Fanuc TP program (LS listing): 190220_hosenrohr_oV5.ls

/PROG  190220_hosenrohr_oV5
/ATTR
COMMENT	= "19-02-22 10:03:29";
PROG_SIZE	= 0;
DEFAULT_GROUP	= 1, 1, *, *, *;
/APPL
    ARC Welding Equipment: 1, *, *, *, *;
/MN
   1:  CALL HOME_ALL;
   1:  UFRAME_NUM = 1;
   1:  UTOOL_NUM = 3;
   1:  COL GUARD ADJUST 150;
   1:  ! -- Layer/Ebene 207 -- !;
   1:  PR[91] = PR[90];
   1:  PR[GP1:91,1] = PR[GP1:90,1] + -0.916;
   1:  PR[GP1:91,2] = PR[GP1:90,2] + 48.907;
   1:  PR[GP1:91,3] = PR[GP1:90,3] + 126.575;
   1:  !Sicherheitspunkt!;
   1:  PR[92] = PR[91];
   1:  PR[92] = PR[GP1:92,3] + 50;
   1:J PR[92];
   1:  !Schweissanfang anfahren!;
   1:L PR[91] R[100]mm/sec CNT100;
   1:  CALL LASER_DRAHT_START;
   1:  PR[GP1:91,1] = PR[GP1:90,1] + -12.234;
   1:  PR[GP1:91,2] = PR[GP1:90,2] + 47.505;
   1:L PR[91] R[100]mm/sec CNT100;
   1:  PR[GP1:91,1] = PR[GP1:90,1] + -13.167;
   1:  PR[GP1:91,2] = PR[GP1:90,2] + 47.191;
   1:L PR[91] R[100]mm/sec CNT100;
   1:  PR[GP1:91,1] = PR[GP1:90,1] + -23.762;
   1:  PR[GP1:91,2] = PR[GP1:90,2] + 43.085;
   1:L PR[91] R[100]mm/sec CNT100;
   1:  PR[GP1:91,1] = PR[GP1:90,1] + -24.573;
   1:  PR[GP1:91,2] = PR[GP1:90,2] + 42.437;
   1:L PR[91] R[100]mm/sec CNT100;
   1:  PR[GP1:91,1] = PR[GP1:90,1] + -33.854;
   1:  PR[GP1:91,2] = PR[GP1:90,2] + 35.865;
   1:L PR[91] R[100]mm/sec CNT100;
   1:  PR[GP1:91,1] = PR[GP1:90,1] + -41.983;
   1:  PR[GP1:91,2] = PR[GP1:90,2] + 26.074;
   1:L PR[91] R[100]mm/sec CNT100;
   1:  PR[GP1:91,1] = PR[GP1:90,1] + -42.514;
   1:  PR[GP1:91,2] = PR[GP1:90,2] + 25.188;
   1:L PR[91] R[100]mm/sec CNT100;
   1:  PR[GP1:91,1] = PR[GP1:90,1] + -47.649;
   1:  PR[GP1:91,2] = PR[GP1:90,2] + 13.555;
   1:L PR[91] R[100]mm/sec CNT100;
   1:  PR[GP1:91,1] = PR[GP1:90,1] + -47.838;
   1:  PR[GP1:91,2] = PR[GP1:90,2] + 12.520;
   1:L PR[91] R[100]mm/sec CNT100;
   1:  PR[GP1:91,1] = PR[GP1:90,1] + -49.592;
   1:  PR[GP1:91,2] = PR[GP1:90,2] + -0.059;
   1:L PR[91] R[100]mm/sec CNT100;
   1:  PR[GP1:91,1] = PR[GP1:90,1] + -49.406;
   1:  PR[GP1:91,2] = PR[GP1:90,2] + -1.079;
   1:L PR[91] R[100]mm/sec CNT100;
   1:  PR[GP1:91,1] = PR[GP1:90,1] + -47.644;
   1:  PR[GP1:91,2] = PR[GP1:90,2] + -13.710;
   1:L PR[91] R[100]mm/sec CNT100;
   1:  PR[GP1:91,1] = PR[GP1:90,1] + -42.514;
   1:  PR[GP1:91,2] = PR[GP1:90,2] + -25.332;
   1:L PR[91] R[100]mm/sec CNT100;
   1:  PR[GP1:91,1] = PR[GP1:90,1] + -41.983;
   1:  PR[GP1:91,2] = PR[GP1:90,2] + -26.218;
   1:L PR[91] R[100]mm/sec CNT100;
   1:  PR[GP1:91,1] = PR[GP1:90,1] + -33.843;
   1:  PR[GP1:91,2] = PR[GP1:90,2] + -36.023;
   1:L PR[91] R[100]mm/sec CNT100;
   1:  PR[GP1:91,1] = PR[GP1:90,1] + -33.064;
   1:  PR[GP1:91,2] = PR[GP1:90,2] + -36.648;
   1:L PR[91] R[100]mm/sec CNT100;
   1:  PR[GP1:91,1] = PR[GP1:90,1] + -23.779;
   1:  PR[GP1:91,2] = PR[GP1:90,2] + -43.223;
   1:L PR[91] R[100]mm/sec CNT100;
   1:  PR[GP1:91,1] = PR[GP1:90,1] + -13.167;
   1:  PR[GP1:91,2] = PR[GP1:90,2] + -47.335;
   1:L PR[91] R[100]mm/sec CNT100;
   1:  PR[GP1:91,1] = PR[GP1:90,1] + -12.234;
   1:  PR[GP1:91,2] = PR[GP1:90,2] + -47.649;
   1:L PR[91] R[100]mm/sec CNT100;
   1:  PR[GP1:91,1] = PR[GP1:90,1] + -0.916;
   1:  PR[GP1:91,2] = PR[GP1:90,2] + -49.051;
   1:L PR[91] R[100]mm/sec CNT100;
   1:  PR[GP1:91,1] = PR[GP1:90,1] + 0.047;
   1:  PR[GP1:91,2] = PR[GP1:90,2] + -49.031;
   1:L PR[91] R[100]mm/sec CNT100;
   1:  PR[GP1:91,1] = PR[GP1:90,1] + 1.125;
   1:  PR[GP1:91,2] = PR[GP1:90,2] + -49.051;
   1:L PR[91] R[100]mm/sec CNT100;
   1:  PR[GP1:91,1] = PR[GP1:90,1] + 12.446;
   1:  PR[GP1:91,2] = PR[GP1:90,2] + -47.650;
   1:L PR[91] R[100]mm/sec CNT100;
   1:  PR[GP1:91,1] = PR[GP1:90,1] + 13.378;
   1:  PR[GP1:91,2] = PR[GP1:90,2] + -47.335;
   1:L PR[91] R[100]mm/sec CNT100;
   1:  PR[GP1:91,1] = PR[GP1:90,1] + 23.975;
   1:  PR[GP1:91,2] = PR[GP1:90,2] + -43.229;
   1:L PR[91] R[100]mm/sec CNT100;
   1:  PR[GP1:91,1] = PR[GP1:90,1] + 24.786;
   1:  PR[GP1:91,2] = PR[GP1:90,2] + -42.581;
   1:L PR[91] R[100]mm/sec CNT100;
   1:  PR[GP1:91,1] = PR[GP1:90,1] + 34.069;
   1:  PR[GP1:91,2] = PR[GP1:90,2] + -36.008;
   1:L PR[91] R[100]mm/sec CNT100;
   1:  PR[GP1:91,1] = PR[GP1:90,1] + 42.197;
   1:  PR[GP1:91,2] = PR[GP1:90,2] + -26.217;
   1:L PR[91] R[100]mm/sec CNT100;
   1:  PR[GP1:91,1] = PR[GP1:90,1] + 42.727;
   1:  PR[GP1:91,2] = PR[GP1:90,2] + -25.331;
   1:L PR[91] R[100]mm/sec CNT100;
   1:  PR[GP1:91,1] = PR[GP1:90,1] + 47.863;
   1:  PR[GP1:91,2] = PR[GP1:90,2] + -13.699;
   1:L PR[91] R[100]mm/sec CNT100;
   1:  PR[GP1:91,1] = PR[GP1:90,1] + 48.051;
   1:  PR[GP1:91,2] = PR[GP1:90,2] + -12.663;
   1:L PR[91] R[100]mm/sec CNT100;
   1:  PR[GP1:91,1] = PR[GP1:90,1] + 49.806;
   1:  PR[GP1:91,2] = PR[GP1:90,2] + -0.085;
   1:L PR[91] R[100]mm/sec CNT100;
   1:  PR[GP1:91,1] = PR[GP1:90,1] + 49.619;
   1:  PR[GP1:91,2] = PR[GP1:90,2] + 0.935;
   1:L PR[91] R[100]mm/sec CNT100;
   1:  PR[GP1:91,1] = PR[GP1:90,1] + 47.857;
   1:  PR[GP1:91,2] = PR[GP1:90,2] + 13.566;
   1:L PR[91] R[100]mm/sec CNT100;
   1:  PR[GP1:91,1] = PR[GP1:90,1] + 42.727;
   1:  PR[GP1:91,2] = PR[GP1:90,2] + 25.187;
   1:L PR[91] R[100]mm/sec CNT100;
   1:  PR[GP1:91,1] = PR[GP1:90,1] + 42.197;
   1:  PR[GP1:91,2] = PR[GP1:90,2] + 26.073;
   1:L PR[91] R[100]mm/sec CNT100;
   1:  PR[GP1:91,1] = PR[GP1:90,1] + 34.058;
   1:  PR[GP1:91,2] = PR[GP1:90,2] + 35.878;
   1:L PR[91] R[100]mm/sec CNT100;
   1:  PR[GP1:91,1] = PR[GP1:90,1] + 33.278;
   1:  PR[GP1:91,2] = PR[GP1:90,2] + 36.503;
   1:L PR[91] R[100]mm/sec CNT100;
   1:  PR[GP1:91,1] = PR[GP1:90,1] + 23.992;
   1:  PR[GP1:91,2] = PR[GP1:90,2] + 43.079;
   1:L PR[91] R[100]mm/sec CNT100;
   1:  PR[GP1:91,1] = PR[GP1:90,1] + 13.378;
   1:  PR[GP1:91,2] = PR[GP1:90,2] + 47.192;
   1:L PR[91] R[100]mm/sec CNT100;
   1:  PR[GP1:91,1] = PR[GP1:90,1] + 12.445;
   1:  PR[GP1:91,2] = PR[GP1:90,2] + 47.506;
   1:L PR[91] R[100]mm/sec CNT100;
   1:  PR[GP1:91,1] = PR[GP1:90,1] + 1.125;
   1:  PR[GP1:91,2] = PR[GP1:90,2] + 48.907;
   1:L PR[91] R[100]mm/sec CNT100;
   1:  PR[GP1:91,1] = PR[GP1:90,1] + 0.047;
   1:  PR[GP1:91,2] = PR[GP1:90,2] + 48.887;
   1:L PR[91] R[100]mm/sec CNT100;
   1:  ! -- Layer/Ebene 208 -- !;
   1:  PR[91] = PR[90];
   1:  PR[GP1:91,1] = PR[GP1:90,1] + -0.545;
   1:  PR[GP1:91,2] = PR[GP1:90,2] + 49.055;
   1:  PR[GP1:91,3] = PR[GP1:90,3] + 127.185;
   1:L PR[91] R[100]mm/sec CNT100;
   1:  PR[GP1:91,1] = PR[GP1:90,1] + -12.137;
   1:  PR[GP1:91,2] = PR[GP1:90,2] + 47.619;
   1:L PR[91] R[100]mm/sec CNT100;
   1:  PR[GP1:91,1] = PR[GP1:90,1] + -12.717;
   1:  PR[GP1:91,2] = PR[GP1:90,2] + 47.424;
   1:L PR[91] R[100]mm/sec CNT100;
   1:  PR[GP1:91,1] = PR[GP1:90,1] + -23.582;
   1:  PR[GP1:91,2] = PR[GP1:90,2] + 43.214;
   1:L PR[91] R[100]mm/sec CNT100;
   1:  PR[GP1:91,1] = PR[GP1:90,1] + -24.086;
   1:  PR[GP1:91,2] = PR[GP1:90,2] + 42.811;
   1:L PR[91] R[100]mm/sec CNT100;
   1:  PR[GP1:91,1] = PR[GP1:90,1] + -33.614;
   1:  PR[GP1:91,2] = PR[GP1:90,2] + 36.064;
   1:L PR[91] R[100]mm/sec CNT100;
   1:  PR[GP1:91,1] = PR[GP1:90,1] + -41.959;
   1:  PR[GP1:91,2] = PR[GP1:90,2] + 26.012;
   1:L PR[91] R[100]mm/sec CNT100;
   1:  PR[GP1:91,1] = PR[GP1:90,1] + -42.288;
   1:  PR[GP1:91,2] = PR[GP1:90,2] + 25.463;
   1:L PR[91] R[100]mm/sec CNT100;
   1:  PR[GP1:91,1] = PR[GP1:90,1] + -47.564;
   1:  PR[GP1:91,2] = PR[GP1:90,2] + 13.512;
   1:L PR[91] R[100]mm/sec CNT100;
   1:  PR[GP1:91,1] = PR[GP1:90,1] + -47.681;
   1:  PR[GP1:91,2] = PR[GP1:90,2] + 12.871;
   1:L PR[91] R[100]mm/sec CNT100;
   1:  PR[GP1:91,1] = PR[GP1:90,1] + -49.484;
   1:  PR[GP1:91,2] = PR[GP1:90,2] + -0.059;
   1:L PR[91] R[100]mm/sec CNT100;
   1:  PR[GP1:91,1] = PR[GP1:90,1] + -49.369;
   1:  PR[GP1:91,2] = PR[GP1:90,2] + -0.690;
   1:L PR[91] R[100]mm/sec CNT100;
   1:  PR[GP1:91,1] = PR[GP1:90,1] + -47.559;
   1:  PR[GP1:91,2] = PR[GP1:90,2] + -13.667;
   1:L PR[91] R[100]mm/sec CNT100;
   1:  PR[GP1:91,1] = PR[GP1:90,1] + -42.288;
   1:  PR[GP1:91,2] = PR[GP1:90,2] + -25.607;
   1:L PR[91] R[100]mm/sec CNT100;
   1:  PR[GP1:91,1] = PR[GP1:90,1] + -41.959;
   1:  PR[GP1:91,2] = PR[GP1:90,2] + -26.156;
   1:L PR[91] R[100]mm/sec CNT100;
   1:  PR[GP1:91,1] = PR[GP1:90,1] + -33.602;
   1:  PR[GP1:91,2] = PR[GP1:90,2] + -36.222;
   1:L PR[91] R[100]mm/sec CNT100;
   1:  PR[GP1:91,1] = PR[GP1:90,1] + -33.120;
   1:  PR[GP1:91,2] = PR[GP1:90,2] + -36.609;
   1:L PR[91] R[100]mm/sec CNT100;
   1:  PR[GP1:91,1] = PR[GP1:90,1] + -23.599;
   1:  PR[GP1:91,2] = PR[GP1:90,2] + -43.351;
   1:L PR[91] R[100]mm/sec CNT100;
   1:  PR[GP1:91,1] = PR[GP1:90,1] + -12.717;
   1:  PR[GP1:91,2] = PR[GP1:90,2] + -47.568;
   1:L PR[91] R[100]mm/sec CNT100;
   1:  PR[GP1:91,1] = PR[GP1:90,1] + -12.138;
   1:  PR[GP1:91,2] = PR[GP1:90,2] + -47.763;
   1:L PR[91] R[100]mm/sec CNT100;
   1:  PR[GP1:91,1] = PR[GP1:90,1] + -0.545;
   1:  PR[GP1:91,2] = PR[GP1:90,2] + -49.199;
   1:L PR[91] R[100]mm/sec CNT100;
   1:  PR[GP1:91,1] = PR[GP1:90,1] + 0.067;
   1:  PR[GP1:91,2] = PR[GP1:90,2] + -49.186;
   1:L PR[91] R[100]mm/sec CNT100;
   1:  PR[GP1:91,1] = PR[GP1:90,1] + 0.754;
   1:  PR[GP1:91,2] = PR[GP1:90,2] + -49.199;
   1:L PR[91] R[100]mm/sec CNT100;
   1:  PR[GP1:91,1] = PR[GP1:90,1] + 12.349;
   1:  PR[GP1:91,2] = PR[GP1:90,2] + -47.764;
   1:L PR[91] R[100]mm/sec CNT100;
   1:  PR[GP1:91,1] = PR[GP1:90,1] + 12.928;
   1:  PR[GP1:91,2] = PR[GP1:90,2] + -47.569;
   1:L PR[91] R[100]mm/sec CNT100;
   1:  PR[GP1:91,1] = PR[GP1:90,1] + 23.795;
   1:  PR[GP1:91,2] = PR[GP1:90,2] + -43.358;
   1:L PR[91] R[100]mm/sec CNT100;
   1:  PR[GP1:91,1] = PR[GP1:90,1] + 24.299;
   1:  PR[GP1:91,2] = PR[GP1:90,2] + -42.955;
   1:L PR[91] R[100]mm/sec CNT100;
   1:  PR[GP1:91,1] = PR[GP1:90,1] + 33.829;
   1:  PR[GP1:91,2] = PR[GP1:90,2] + -36.207;
   1:L PR[91] R[100]mm/sec CNT100;
   1:  PR[GP1:91,1] = PR[GP1:90,1] + 42.173;
   1:  PR[GP1:91,2] = PR[GP1:90,2] + -26.155;
   1:L PR[91] R[100]mm/sec CNT100;
   1:  PR[GP1:91,1] = PR[GP1:90,1] + 42.501;
   1:  PR[GP1:91,2] = PR[GP1:90,2] + -25.607;
   1:L PR[91] R[100]mm/sec CNT100;
   1:  PR[GP1:91,1] = PR[GP1:90,1] + 47.777;
   1:  PR[GP1:91,2] = PR[GP1:90,2] + -13.655;
   1:L PR[91] R[100]mm/sec CNT100;
   1:  PR[GP1:91,1] = PR[GP1:90,1] + 47.894;
   1:  PR[GP1:91,2] = PR[GP1:90,2] + -13.014;
   1:L PR[91] R[100]mm/sec CNT100;
   1:  PR[GP1:91,1] = PR[GP1:90,1] + 49.698;
   1:  PR[GP1:91,2] = PR[GP1:90,2] + -0.085;
   1:L PR[91] R[100]mm/sec CNT100;
   1:  PR[GP1:91,1] = PR[GP1:90,1] + 49.582;
   1:  PR[GP1:91,2] = PR[GP1:90,2] + 0.546;
   1:L PR[91] R[100]mm/sec CNT100;
   1:  PR[GP1:91,1] = PR[GP1:90,1] + 47.772;
   1:  PR[GP1:91,2] = PR[GP1:90,2] + 13.523;
   1:L PR[91] R[100]mm/sec CNT100;
   1:  PR[GP1:91,1] = PR[GP1:90,1] + 42.501;
   1:  PR[GP1:91,2] = PR[GP1:90,2] + 25.463;
   1:L PR[91] R[100]mm/sec CNT100;
   1:  PR[GP1:91,1] = PR[GP1:90,1] + 42.173;
   1:  PR[GP1:91,2] = PR[GP1:90,2] + 26.011;
   1:L PR[91] R[100]mm/sec CNT100;
   1:  PR[GP1:91,1] = PR[GP1:90,1] + 33.817;
   1:  PR[GP1:91,2] = PR[GP1:90,2] + 36.077;
   1:L PR[91] R[100]mm/sec CNT100;
   1:  PR[GP1:91,1] = PR[GP1:90,1] + 33.334;
   1:  PR[GP1:91,2] = PR[GP1:90,2] + 36.464;
   1:L PR[91] R[100]mm/sec CNT100;
   1:  PR[GP1:91,1] = PR[GP1:90,1] + 23.812;
   1:  PR[GP1:91,2] = PR[GP1:90,2] + 43.207;
   1:L PR[91] R[100]mm/sec CNT100;
   1:  PR[GP1:91,1] = PR[GP1:90,1] + 12.928;
   1:  PR[GP1:91,2] = PR[GP1:90,2] + 47.425;
   1:L PR[91] R[100]mm/sec CNT100;
   1:  PR[GP1:91,1] = PR[GP1:90,1] + 12.349;
   1:  PR[GP1:91,2] = PR[GP1:90,2] + 47.620;
   1:L PR[91] R[100]mm/sec CNT100;
   1:  PR[GP1:91,1] = PR[GP1:90,1] + 0.754;
   1:  PR[GP1:91,2] = PR[GP1:90,2] + 49.056;
   1:L PR[91] R[100]mm/sec CNT100;
   1:  PR[GP1:91,1] = PR[GP1:90,1] + 0.067;
   1:  PR[GP1:91,2] = PR[GP1:90,2] + 49.042;
   1:L PR[91] R[100]mm/sec CNT100;
   1:  ! -- Layer/Ebene 209 -- !;
   1:  PR[91] = PR[90];
   1:  PR[GP1:91,1] = PR[GP1:90,1] + -12.041;
   1:  PR[GP1:91,2] = PR[GP1:90,2] + 47.733;
   1:  PR[GP1:91,3] = PR[GP1:90,3] + 127.795;
   1:L PR[91] R[100]mm/sec CNT100;
   1:  PR[GP1:91,1] = PR[GP1:90,1] + -12.266;
   1:  PR[GP1:91,2] = PR[GP1:90,2] + 47.657;
   1:L PR[91] R[100]mm/sec CNT100;
   1:  PR[GP1:91,1] = PR[GP1:90,1] + -23.402;
   1:  PR[GP1:91,2] = PR[GP1:90,2] + 43.342;
   1:L PR[91] R[100]mm/sec CNT100;
   1:  PR[GP1:91,1] = PR[GP1:90,1] + -23.600;
   1:  PR[GP1:91,2] = PR[GP1:90,2] + 43.184;
   1:L PR[91] R[100]mm/sec CNT100;
   1:  PR[GP1:91,1] = PR[GP1:90,1] + -33.373;
   1:  PR[GP1:91,2] = PR[GP1:90,2] + 36.263;
   1:L PR[91] R[100]mm/sec CNT100;
   1:  PR[GP1:91,1] = PR[GP1:90,1] + -41.935;
   1:  PR[GP1:91,2] = PR[GP1:90,2] + 25.950;
   1:L PR[91] R[100]mm/sec CNT100;
   1:  PR[GP1:91,1] = PR[GP1:90,1] + -42.062;
   1:  PR[GP1:91,2] = PR[GP1:90,2] + 25.739;
   1:L PR[91] R[100]mm/sec CNT100;
   1:  PR[GP1:91,1] = PR[GP1:90,1] + -47.479;
   1:  PR[GP1:91,2] = PR[GP1:90,2] + 13.468;
   1:L PR[91] R[100]mm/sec CNT100;
   1:  PR[GP1:91,1] = PR[GP1:90,1] + -47.524;
   1:  PR[GP1:91,2] = PR[GP1:90,2] + 13.221;
   1:L PR[91] R[100]mm/sec CNT100;
   1:  PR[GP1:91,1] = PR[GP1:90,1] + -49.376;
   1:  PR[GP1:91,2] = PR[GP1:90,2] + -0.059;
   1:L PR[91] R[100]mm/sec CNT100;
   1:  PR[GP1:91,1] = PR[GP1:90,1] + -49.332;
   1:  PR[GP1:91,2] = PR[GP1:90,2] + -0.302;
   1:L PR[91] R[100]mm/sec CNT100;
   1:  PR[GP1:91,1] = PR[GP1:90,1] + -47.474;
   1:  PR[GP1:91,2] = PR[GP1:90,2] + -13.624;
   1:L PR[91] R[100]mm/sec CNT100;
   1:  PR[GP1:91,1] = PR[GP1:90,1] + -42.062;
   1:  PR[GP1:91,2] = PR[GP1:90,2] + -25.883;
   1:L PR[91] R[100]mm/sec CNT100;
   1:  PR[GP1:91,1] = PR[GP1:90,1] + -41.935;
   1:  PR[GP1:91,2] = PR[GP1:90,2] + -26.094;
   1:L PR[91] R[100]mm/sec CNT100;
   1:  PR[GP1:91,1] = PR[GP1:90,1] + -33.362;
   1:  PR[GP1:91,2] = PR[GP1:90,2] + -36.421;
   1:L PR[91] R[100]mm/sec CNT100;
   1:  PR[GP1:91,1] = PR[GP1:90,1] + -33.176;
   1:  PR[GP1:91,2] = PR[GP1:90,2] + -36.570;
   1:L PR[91] R[100]mm/sec CNT100;
   1:  PR[GP1:91,1] = PR[GP1:90,1] + -23.418;
   1:  PR[GP1:91,2] = PR[GP1:90,2] + -43.480;
   1:L PR[91] R[100]mm/sec CNT100;
   1:  PR[GP1:91,1] = PR[GP1:90,1] + -12.266;
   1:  PR[GP1:91,2] = PR[GP1:90,2] + -47.801;
   1:L PR[91] R[100]mm/sec CNT100;
   1:  PR[GP1:91,1] = PR[GP1:90,1] + -12.041;
   1:  PR[GP1:91,2] = PR[GP1:90,2] + -47.877;
   1:L PR[91] R[100]mm/sec CNT100;
   1:  PR[GP1:91,1] = PR[GP1:90,1] + -0.168;
   1:  PR[GP1:91,2] = PR[GP1:90,2] + -49.348;
   1:L PR[91] R[100]mm/sec CNT100;
   1:  PR[GP1:91,1] = PR[GP1:90,1] + 0.377;
   1:L PR[91] R[100]mm/sec CNT100;
   1:  PR[GP1:91,1] = PR[GP1:90,1] + 12.252;
   1:  PR[GP1:91,2] = PR[GP1:90,2] + -47.878;
   1:L PR[91] R[100]mm/sec CNT100;
   1:  PR[GP1:91,1] = PR[GP1:90,1] + 12.478;
   1:  PR[GP1:91,2] = PR[GP1:90,2] + -47.802;
   1:L PR[91] R[100]mm/sec CNT100;
   1:  PR[GP1:91,1] = PR[GP1:90,1] + 23.615;
   1:  PR[GP1:91,2] = PR[GP1:90,2] + -43.486;
   1:L PR[91] R[100]mm/sec CNT100;
   1:  PR[GP1:91,1] = PR[GP1:90,1] + 23.812;
   1:  PR[GP1:91,2] = PR[GP1:90,2] + -43.328;
   1:L PR[91] R[100]mm/sec CNT100;
   1:  PR[GP1:91,1] = PR[GP1:90,1] + 33.588;
   1:  PR[GP1:91,2] = PR[GP1:90,2] + -36.406;
   1:L PR[91] R[100]mm/sec CNT100;
   1:  PR[GP1:91,1] = PR[GP1:90,1] + 42.149;
   1:  PR[GP1:91,2] = PR[GP1:90,2] + -26.093;
   1:L PR[91] R[100]mm/sec CNT100;
   1:  PR[GP1:91,1] = PR[GP1:90,1] + 42.275;
   1:  PR[GP1:91,2] = PR[GP1:90,2] + -25.882;
   1:L PR[91] R[100]mm/sec CNT100;
   1:  PR[GP1:91,1] = PR[GP1:90,1] + 47.692;
   1:  PR[GP1:91,2] = PR[GP1:90,2] + -13.612;
   1:L PR[91] R[100]mm/sec CNT100;
   1:  PR[GP1:91,1] = PR[GP1:90,1] + 47.737;
   1:  PR[GP1:91,2] = PR[GP1:90,2] + -13.365;
   1:L PR[91] R[100]mm/sec CNT100;
   1:  PR[GP1:91,1] = PR[GP1:90,1] + 49.589;
   1:  PR[GP1:91,2] = PR[GP1:90,2] + -0.085;
   1:L PR[91] R[100]mm/sec CNT100;
   1:  PR[GP1:91,1] = PR[GP1:90,1] + 49.545;
   1:  PR[GP1:91,2] = PR[GP1:90,2] + 0.158;
   1:L PR[91] R[100]mm/sec CNT100;
   1:  PR[GP1:91,1] = PR[GP1:90,1] + 47.687;
   1:  PR[GP1:91,2] = PR[GP1:90,2] + 13.480;
   1:L PR[91] R[100]mm/sec CNT100;
   1:  PR[GP1:91,1] = PR[GP1:90,1] + 42.275;
   1:  PR[GP1:91,2] = PR[GP1:90,2] + 25.738;
   1:L PR[91] R[100]mm/sec CNT100;
   1:  PR[GP1:91,1] = PR[GP1:90,1] + 42.149;
   1:  PR[GP1:91,2] = PR[GP1:90,2] + 25.949;
   1:L PR[91] R[100]mm/sec CNT100;
   1:  PR[GP1:91,1] = PR[GP1:90,1] + 33.577;
   1:  PR[GP1:91,2] = PR[GP1:90,2] + 36.276;
   1:L PR[91] R[100]mm/sec CNT100;
   1:  PR[GP1:91,1] = PR[GP1:90,1] + 33.390;
   1:  PR[GP1:91,2] = PR[GP1:90,2] + 36.425;
   1:L PR[91] R[100]mm/sec CNT100;
   1:  PR[GP1:91,1] = PR[GP1:90,1] + 23.631;
   1:  PR[GP1:91,2] = PR[GP1:90,2] + 43.336;
   1:L PR[91] R[100]mm/sec CNT100;
   1:  PR[GP1:91,1] = PR[GP1:90,1] + 12.477;
   1:  PR[GP1:91,2] = PR[GP1:90,2] + 47.658;
   1:L PR[91] R[100]mm/sec CNT100;
   1:  PR[GP1:91,1] = PR[GP1:90,1] + 12.252;
   1:  PR[GP1:91,2] = PR[GP1:90,2] + 47.734;
   1:L PR[91] R[100]mm/sec CNT100;
   1:  PR[GP1:91,1] = PR[GP1:90,1] + 0.377;
   1:  PR[GP1:91,2] = PR[GP1:90,2] + 49.204;
   1:L PR[91] R[100]mm/sec CNT100;
   1:  PR[GP1:91,1] = PR[GP1:90,1] + -0.168;
   1:L PR[91] R[100]mm/sec CNT100;
   1:  ! -- Layer/Ebene 210 -- !;
   1:  PR[91] = PR[90];
   1:  PR[GP1:91,1] = PR[GP1:90,1] + -11.979;
   1:  PR[GP1:91,2] = PR[GP1:90,2] + 47.821;
   1:  PR[GP1:91,3] = PR[GP1:90,3] + 128.405;
   1:L PR[91] R[100]mm/sec CNT100;
   1:  PR[GP1:91,1] = PR[GP1:90,1] + -23.226;
   1:  PR[GP1:91,2] = PR[GP1:90,2] + 43.462;
   1:L PR[91] R[100]mm/sec CNT100;
   1:  PR[GP1:91,1] = PR[GP1:90,1] + -23.300;
   1:  PR[GP1:91,2] = PR[GP1:90,2] + 43.425;
   1:L PR[91] R[100]mm/sec CNT100;
   1:  PR[GP1:91,1] = PR[GP1:90,1] + -33.152;
   1:  PR[GP1:91,2] = PR[GP1:90,2] + 36.449;
   1:L PR[91] R[100]mm/sec CNT100;
   1:  PR[GP1:91,1] = PR[GP1:90,1] + -33.209;
   1:  PR[GP1:91,2] = PR[GP1:90,2] + 36.392;
   1:L PR[91] R[100]mm/sec CNT100;
   1:  PR[GP1:91,1] = PR[GP1:90,1] + -41.871;
   1:  PR[GP1:91,2] = PR[GP1:90,2] + 25.958;
   1:L PR[91] R[100]mm/sec CNT100;
   1:  PR[GP1:91,1] = PR[GP1:90,1] + -47.397;
   1:  PR[GP1:91,2] = PR[GP1:90,2] + 13.461;
   1:L PR[91] R[100]mm/sec CNT100;
   1:  PR[GP1:91,1] = PR[GP1:90,1] + -49.288;
   1:  PR[GP1:91,2] = PR[GP1:90,2] + -0.072;
   1:L PR[91] R[100]mm/sec CNT100;
   1:  PR[GP1:91,1] = PR[GP1:90,1] + -47.411;
   1:  PR[GP1:91,2] = PR[GP1:90,2] + -13.529;
   1:L PR[91] R[100]mm/sec CNT100;
   1:  PR[GP1:91,1] = PR[GP1:90,1] + -47.399;
   1:  PR[GP1:91,2] = PR[GP1:90,2] + -13.600;
   1:L PR[91] R[100]mm/sec CNT100;
   1:  PR[GP1:91,1] = PR[GP1:90,1] + -41.871;
   1:  PR[GP1:91,2] = PR[GP1:90,2] + -26.102;
   1:L PR[91] R[100]mm/sec CNT100;
   1:  PR[GP1:91,1] = PR[GP1:90,1] + -33.209;
   1:  PR[GP1:91,2] = PR[GP1:90,2] + -36.536;
   1:L PR[91] R[100]mm/sec CNT100;
   1:  PR[GP1:91,1] = PR[GP1:90,1] + -33.152;
   1:  PR[GP1:91,2] = PR[GP1:90,2] + -36.592;
   1:L PR[91] R[100]mm/sec CNT100;
   1:  PR[GP1:91,1] = PR[GP1:90,1] + -23.300;
   1:  PR[GP1:91,2] = PR[GP1:90,2] + -43.569;
   1:L PR[91] R[100]mm/sec CNT100;
   1:  PR[GP1:91,1] = PR[GP1:90,1] + -23.226;
   1:  PR[GP1:91,2] = PR[GP1:90,2] + -43.606;
   1:L PR[91] R[100]mm/sec CNT100;
   1:  PR[GP1:91,1] = PR[GP1:90,1] + -11.979;
   1:  PR[GP1:91,2] = PR[GP1:90,2] + -47.965;
   1:L PR[91] R[100]mm/sec CNT100;
   1:  PR[GP1:91,1] = PR[GP1:90,1] + 0.105;
   1:  PR[GP1:91,2] = PR[GP1:90,2] + -49.467;
   1:L PR[91] R[100]mm/sec CNT100;
   1:  PR[GP1:91,1] = PR[GP1:90,1] + 12.190;
   1:  PR[GP1:91,2] = PR[GP1:90,2] + -47.965;
   1:L PR[91] R[100]mm/sec CNT100;
   1:  PR[GP1:91,1] = PR[GP1:90,1] + 23.439;
   1:  PR[GP1:91,2] = PR[GP1:90,2] + -43.606;
   1:L PR[91] R[100]mm/sec CNT100;
   1:  PR[GP1:91,1] = PR[GP1:90,1] + 23.513;
   1:  PR[GP1:91,2] = PR[GP1:90,2] + -43.569;
   1:L PR[91] R[100]mm/sec CNT100;
   1:  PR[GP1:91,1] = PR[GP1:90,1] + 33.367;
   1:  PR[GP1:91,2] = PR[GP1:90,2] + -36.591;
   1:L PR[91] R[100]mm/sec CNT100;
   1:  PR[GP1:91,1] = PR[GP1:90,1] + 33.421;
   1:  PR[GP1:91,2] = PR[GP1:90,2] + -36.536;
   1:L PR[91] R[100]mm/sec CNT100;
   1:  PR[GP1:91,1] = PR[GP1:90,1] + 42.085;
   1:  PR[GP1:91,2] = PR[GP1:90,2] + -26.101;
   1:L PR[91] R[100]mm/sec CNT100;
   1:  PR[GP1:91,1] = PR[GP1:90,1] + 47.610;
   1:  PR[GP1:91,2] = PR[GP1:90,2] + -13.605;
   1:L PR[91] R[100]mm/sec CNT100;
   1:  PR[GP1:91,1] = PR[GP1:90,1] + 49.501;
   1:  PR[GP1:91,2] = PR[GP1:90,2] + -0.072;
   1:L PR[91] R[100]mm/sec CNT100;
   1:  PR[GP1:91,1] = PR[GP1:90,1] + 47.610;
   1:  PR[GP1:91,2] = PR[GP1:90,2] + 13.461;
   1:L PR[91] R[100]mm/sec CNT100;
   1:  PR[GP1:91,1] = PR[GP1:90,1] + 42.085;
   1:  PR[GP1:91,2] = PR[GP1:90,2] + 25.957;
   1:L PR[91] R[100]mm/sec CNT100;
   1:  PR[GP1:91,1] = PR[GP1:90,1] + 33.421;
   1:  PR[GP1:91,2] = PR[GP1:90,2] + 36.393;
   1:L PR[91] R[100]mm/sec CNT100;
   1:  PR[GP1:91,1] = PR[GP1:90,1] + 33.367;
   1:  PR[GP1:91,2] = PR[GP1:90,2] + 36.447;
   1:L PR[91] R[100]mm/sec CNT100;
   1:  PR[GP1:91,1] = PR[GP1:90,1] + 23.513;
   1:  PR[GP1:91,2] = PR[GP1:90,2] + 43.425;
   1:L PR[91] R[100]mm/sec CNT100;
   1:  PR[GP1:91,1] = PR[GP1:90,1] + 23.439;
   1:  PR[GP1:91,2] = PR[GP1:90,2] + 43.462;
   1:L PR[91] R[100]mm/sec CNT100;
   1:  PR[GP1:91,1] = PR[GP1:90,1] + 12.181;
   1:  PR[GP1:91,2] = PR[GP1:90,2] + 47.825;
   1:L PR[91] R[100]mm/sec CNT100;
   1:  PR[GP1:91,1] = PR[GP1:90,1] + 12.099;
   1:  PR[GP1:91,2] = PR[GP1:90,2] + 47.838;
   1:L PR[91] R[100]mm/sec CNT100;
   1:  PR[GP1:91,1] = PR[GP1:90,1] + 0.105;
   1:  PR[GP1:91,2] = PR[GP1:90,2] + 49.323;
   1:L PR[91] R[100]mm/sec CNT100;
   1:  ! -- Layer/Ebene 211 -- !;
   1:  PR[91] = PR[90];
   1:  PR[GP1:91,1] = PR[GP1:90,1] + -11.144;
   1:  PR[GP1:91,2] = PR[GP1:90,2] + 47.930;
   1:  PR[GP1:91,3] = PR[GP1:90,3] + 129.015;
   1:L PR[91] R[100]mm/sec CNT100;
   1:  PR[GP1:91,1] = PR[GP1:90,1] + -12.168;
   1:  PR[GP1:91,2] = PR[GP1:90,2] + 47.768;
   1:L PR[91] R[100]mm/sec CNT100;
   1:  PR[GP1:91,1] = PR[GP1:90,1] + -22.726;
   1:  PR[GP1:91,2] = PR[GP1:90,2] + 43.676;
   1:L PR[91] R[100]mm/sec CNT100;
   1:  PR[GP1:91,1] = PR[GP1:90,1] + -23.649;
   1:  PR[GP1:91,2] = PR[GP1:90,2] + 43.205;
   1:L PR[91] R[100]mm/sec CNT100;
   1:  PR[GP1:91,1] = PR[GP1:90,1] + -32.890;
   1:  PR[GP1:91,2] = PR[GP1:90,2] + 36.662;
   1:L PR[91] R[100]mm/sec CNT100;
   1:  PR[GP1:91,1] = PR[GP1:90,1] + -33.621;
   1:  PR[GP1:91,2] = PR[GP1:90,2] + 35.931;
   1:L PR[91] R[100]mm/sec CNT100;
   1:  PR[GP1:91,1] = PR[GP1:90,1] + -41.756;
   1:  PR[GP1:91,2] = PR[GP1:90,2] + 26.132;
   1:L PR[91] R[100]mm/sec CNT100;
   1:  PR[GP1:91,1] = PR[GP1:90,1] + -42.222;
   1:  PR[GP1:91,2] = PR[GP1:90,2] + 25.217;
   1:L PR[91] R[100]mm/sec CNT100;
   1:  PR[GP1:91,1] = PR[GP1:90,1] + -47.364;
   1:  PR[GP1:91,2] = PR[GP1:90,2] + 13.569;
   1:L PR[91] R[100]mm/sec CNT100;
   1:  PR[GP1:91,1] = PR[GP1:90,1] + -49.126;
   1:  PR[GP1:91,2] = PR[GP1:90,2] + 0.936;
   1:L PR[91] R[100]mm/sec CNT100;
   1:  PR[GP1:91,1] = PR[GP1:90,1] + -49.287;
   1:  PR[GP1:91,2] = PR[GP1:90,2] + -0.078;
   1:L PR[91] R[100]mm/sec CNT100;
   1:  PR[GP1:91,1] = PR[GP1:90,1] + -47.527;
   1:  PR[GP1:91,2] = PR[GP1:90,2] + -12.694;
   1:L PR[91] R[100]mm/sec CNT100;
   1:  PR[GP1:91,1] = PR[GP1:90,1] + -47.366;
   1:  PR[GP1:91,2] = PR[GP1:90,2] + -13.708;
   1:L PR[91] R[100]mm/sec CNT100;
   1:  PR[GP1:91,1] = PR[GP1:90,1] + -42.222;
   1:  PR[GP1:91,2] = PR[GP1:90,2] + -25.361;
   1:L PR[91] R[100]mm/sec CNT100;
   1:  PR[GP1:91,1] = PR[GP1:90,1] + -41.756;
   1:  PR[GP1:91,2] = PR[GP1:90,2] + -26.276;
   1:L PR[91] R[100]mm/sec CNT100;
   1:  PR[GP1:91,1] = PR[GP1:90,1] + -33.621;
   1:  PR[GP1:91,2] = PR[GP1:90,2] + -36.075;
   1:L PR[91] R[100]mm/sec CNT100;
   1:  PR[GP1:91,1] = PR[GP1:90,1] + -32.890;
   1:  PR[GP1:91,2] = PR[GP1:90,2] + -36.806;
   1:L PR[91] R[100]mm/sec CNT100;
   1:  PR[GP1:91,1] = PR[GP1:90,1] + -23.649;
   1:  PR[GP1:91,2] = PR[GP1:90,2] + -43.349;
   1:L PR[91] R[100]mm/sec CNT100;
   1:  PR[GP1:91,1] = PR[GP1:90,1] + -22.726;
   1:  PR[GP1:91,2] = PR[GP1:90,2] + -43.820;
   1:L PR[91] R[100]mm/sec CNT100;
   1:  PR[GP1:91,1] = PR[GP1:90,1] + -12.177;
   1:  PR[GP1:91,2] = PR[GP1:90,2] + -47.908;
   1:L PR[91] R[100]mm/sec CNT100;
   1:  PR[GP1:91,1] = PR[GP1:90,1] + -0.909;
   1:  PR[GP1:91,2] = PR[GP1:90,2] + -49.304;
   1:L PR[91] R[100]mm/sec CNT100;
   1:  PR[GP1:91,1] = PR[GP1:90,1] + 0.115;
   1:  PR[GP1:91,2] = PR[GP1:90,2] + -49.466;
   1:L PR[91] R[100]mm/sec CNT100;
   1:  PR[GP1:91,1] = PR[GP1:90,1] + 11.355;
   1:  PR[GP1:91,2] = PR[GP1:90,2] + -48.074;
   1:L PR[91] R[100]mm/sec CNT100;
   1:  PR[GP1:91,1] = PR[GP1:90,1] + 12.379;
   1:  PR[GP1:91,2] = PR[GP1:90,2] + -47.912;
   1:L PR[91] R[100]mm/sec CNT100;
   1:  PR[GP1:91,1] = PR[GP1:90,1] + 22.938;
   1:  PR[GP1:91,2] = PR[GP1:90,2] + -43.820;
   1:L PR[91] R[100]mm/sec CNT100;
   1:  PR[GP1:91,1] = PR[GP1:90,1] + 23.862;
   1:  PR[GP1:91,2] = PR[GP1:90,2] + -43.350;
   1:L PR[91] R[100]mm/sec CNT100;
   1:  PR[GP1:91,1] = PR[GP1:90,1] + 33.105;
   1:  PR[GP1:91,2] = PR[GP1:90,2] + -36.805;
   1:L PR[91] R[100]mm/sec CNT100;
   1:  PR[GP1:91,1] = PR[GP1:90,1] + 33.834;
   1:  PR[GP1:91,2] = PR[GP1:90,2] + -36.076;
   1:L PR[91] R[100]mm/sec CNT100;
   1:  PR[GP1:91,1] = PR[GP1:90,1] + 41.970;
   1:  PR[GP1:91,2] = PR[GP1:90,2] + -26.275;
   1:L PR[91] R[100]mm/sec CNT100;
   1:  PR[GP1:91,1] = PR[GP1:90,1] + 42.436;
   1:  PR[GP1:91,2] = PR[GP1:90,2] + -25.360;
   1:L PR[91] R[100]mm/sec CNT100;
   1:  PR[GP1:91,1] = PR[GP1:90,1] + 47.578;
   1:  PR[GP1:91,2] = PR[GP1:90,2] + -13.713;
   1:L PR[91] R[100]mm/sec CNT100;
   1:  PR[GP1:91,1] = PR[GP1:90,1] + 49.339;
   1:  PR[GP1:91,2] = PR[GP1:90,2] + -1.080;
   1:L PR[91] R[100]mm/sec CNT100;
   1:  PR[GP1:91,1] = PR[GP1:90,1] + 49.500;
   1:  PR[GP1:91,2] = PR[GP1:90,2] + -0.066;
   1:L PR[91] R[100]mm/sec CNT100;
   1:  PR[GP1:91,1] = PR[GP1:90,1] + 47.740;
   1:  PR[GP1:91,2] = PR[GP1:90,2] + 12.550;
   1:L PR[91] R[100]mm/sec CNT100;
   1:  PR[GP1:91,1] = PR[GP1:90,1] + 47.580;
   1:  PR[GP1:91,2] = PR[GP1:90,2] + 13.564;
   1:L PR[91] R[100]mm/sec CNT100;
   1:  PR[GP1:91,1] = PR[GP1:90,1] + 42.436;
   1:  PR[GP1:91,2] = PR[GP1:90,2] + 25.216;
   1:L PR[91] R[100]mm/sec CNT100;
   1:  PR[GP1:91,1] = PR[GP1:90,1] + 41.970;
   1:  PR[GP1:91,2] = PR[GP1:90,2] + 26.131;
   1:L PR[91] R[100]mm/sec CNT100;
   1:  PR[GP1:91,1] = PR[GP1:90,1] + 33.834;
   1:  PR[GP1:91,2] = PR[GP1:90,2] + 35.932;
   1:L PR[91] R[100]mm/sec CNT100;
   1:  PR[GP1:91,1] = PR[GP1:90,1] + 33.105;
   1:  PR[GP1:91,2] = PR[GP1:90,2] + 36.661;
   1:L PR[91] R[100]mm/sec CNT100;
   1:  PR[GP1:91,1] = PR[GP1:90,1] + 23.862;
   1:  PR[GP1:91,2] = PR[GP1:90,2] + 43.206;
   1:L PR[91] R[100]mm/sec CNT100;
   1:  PR[GP1:91,1] = PR[GP1:90,1] + 22.938;
   1:  PR[GP1:91,2] = PR[GP1:90,2] + 43.676;
   1:L PR[91] R[100]mm/sec CNT100;
   1:  PR[GP1:91,1] = PR[GP1:90,1] + 12.379;
   1:  PR[GP1:91,2] = PR[GP1:90,2] + 47.768;
   1:L PR[91] R[100]mm/sec CNT100;
   1:  PR[GP1:91,1] = PR[GP1:90,1] + 11.355;
   1:  PR[GP1:91,2] = PR[GP1:90,2] + 47.930;
   1:L PR[91] R[100]mm/sec CNT100;
   1:  PR[GP1:91,1] = PR[GP1:90,1] + 0.105;
   1:  PR[GP1:91,2] = PR[GP1:90,2] + 49.323;
   1:L PR[91] R[100]mm/sec CNT100;
   1:  ! -- Layer/Ebene 212 -- !;
   1:  PR[91] = PR[90];
   1:  PR[GP1:91,1] = PR[GP1:90,1] + -10.400;
   1:  PR[GP1:91,2] = PR[GP1:90,2] + 48.022;
   1:  PR[GP1:91,3] = PR[GP1:90,3] + 129.625;
   1:L PR[91] R[100]mm/sec CNT100;
   1:  PR[GP1:91,1] = PR[GP1:90,1] + -12.366;
   1:  PR[GP1:91,2] = PR[GP1:90,2] + 47.710;
   1:L PR[91] R[100]mm/sec CNT100;
   1:  PR[GP1:91,1] = PR[GP1:90,1] + -22.225;
   1:  PR[GP1:91,2] = PR[GP1:90,2] + 43.890;
   1:L PR[91] R[100]mm/sec CNT100;
   1:  PR[GP1:91,1] = PR[GP1:90,1] + -23.999;
   1:  PR[GP1:91,2] = PR[GP1:90,2] + 42.986;
   1:L PR[91] R[100]mm/sec CNT100;
   1:  PR[GP1:91,1] = PR[GP1:90,1] + -32.627;
   1:  PR[GP1:91,2] = PR[GP1:90,2] + 36.876;
   1:L PR[91] R[100]mm/sec CNT100;
   1:  PR[GP1:91,1] = PR[GP1:90,1] + -34.033;
   1:  PR[GP1:91,2] = PR[GP1:90,2] + 35.470;
   1:L PR[91] R[100]mm/sec CNT100;
   1:  PR[GP1:91,1] = PR[GP1:90,1] + -41.630;
   1:  PR[GP1:91,2] = PR[GP1:90,2] + 26.319;
   1:L PR[91] R[100]mm/sec CNT100;
   1:  PR[GP1:91,1] = PR[GP1:90,1] + -42.529;
   1:  PR[GP1:91,2] = PR[GP1:90,2] + 24.554;
   1:L PR[91] R[100]mm/sec CNT100;
   1:  PR[GP1:91,1] = PR[GP1:90,1] + -47.331;
   1:  PR[GP1:91,2] = PR[GP1:90,2] + 13.677;
   1:L PR[91] R[100]mm/sec CNT100;
   1:  PR[GP1:91,1] = PR[GP1:90,1] + -48.977;
   1:  PR[GP1:91,2] = PR[GP1:90,2] + 1.879;
   1:L PR[91] R[100]mm/sec CNT100;
   1:  PR[GP1:91,1] = PR[GP1:90,1] + -49.287;
   1:  PR[GP1:91,2] = PR[GP1:90,2] + -0.078;
   1:L PR[91] R[100]mm/sec CNT100;
   1:  PR[GP1:91,1] = PR[GP1:90,1] + -47.643;
   1:  PR[GP1:91,2] = PR[GP1:90,2] + -11.860;
   1:L PR[91] R[100]mm/sec CNT100;
   1:  PR[GP1:91,1] = PR[GP1:90,1] + -47.334;
   1:  PR[GP1:91,2] = PR[GP1:90,2] + -13.816;
   1:L PR[91] R[100]mm/sec CNT100;
   1:  PR[GP1:91,1] = PR[GP1:90,1] + -42.530;
   1:  PR[GP1:91,2] = PR[GP1:90,2] + -24.698;
   1:L PR[91] R[100]mm/sec CNT100;
   1:  PR[GP1:91,1] = PR[GP1:90,1] + -41.630;
   1:  PR[GP1:91,2] = PR[GP1:90,2] + -26.463;
   1:L PR[91] R[100]mm/sec CNT100;
   1:  PR[GP1:91,1] = PR[GP1:90,1] + -34.033;
   1:  PR[GP1:91,2] = PR[GP1:90,2] + -35.614;
   1:L PR[91] R[100]mm/sec CNT100;
   1:  PR[GP1:91,1] = PR[GP1:90,1] + -32.627;
   1:  PR[GP1:91,2] = PR[GP1:90,2] + -37.020;
   1:L PR[91] R[100]mm/sec CNT100;
   1:  PR[GP1:91,1] = PR[GP1:90,1] + -23.999;
   1:  PR[GP1:91,2] = PR[GP1:90,2] + -43.130;
   1:L PR[91] R[100]mm/sec CNT100;
   1:  PR[GP1:91,1] = PR[GP1:90,1] + -22.225;
   1:  PR[GP1:91,2] = PR[GP1:90,2] + -44.034;
   1:L PR[91] R[100]mm/sec CNT100;
   1:  PR[GP1:91,1] = PR[GP1:90,1] + -12.376;
   1:  PR[GP1:91,2] = PR[GP1:90,2] + -47.851;
   1:L PR[91] R[100]mm/sec CNT100;
   1:  PR[GP1:91,1] = PR[GP1:90,1] + -1.851;
   1:  PR[GP1:91,2] = PR[GP1:90,2] + -49.155;
   1:L PR[91] R[100]mm/sec CNT100;
   1:  PR[GP1:91,1] = PR[GP1:90,1] + 0.115;
   1:  PR[GP1:91,2] = PR[GP1:90,2] + -49.466;
   1:L PR[91] R[100]mm/sec CNT100;
   1:  PR[GP1:91,1] = PR[GP1:90,1] + 10.611;
   1:  PR[GP1:91,2] = PR[GP1:90,2] + -48.166;
   1:L PR[91] R[100]mm/sec CNT100;
   1:  PR[GP1:91,1] = PR[GP1:90,1] + 12.577;
   1:  PR[GP1:91,2] = PR[GP1:90,2] + -47.855;
   1:L PR[91] R[100]mm/sec CNT100;
   1:  PR[GP1:91,1] = PR[GP1:90,1] + 22.438;
   1:  PR[GP1:91,2] = PR[GP1:90,2] + -44.034;
   1:L PR[91] R[100]mm/sec CNT100;
   1:  PR[GP1:91,1] = PR[GP1:90,1] + 24.212;
   1:  PR[GP1:91,2] = PR[GP1:90,2] + -43.130;
   1:L PR[91] R[100]mm/sec CNT100;
   1:  PR[GP1:91,1] = PR[GP1:90,1] + 32.842;
   1:  PR[GP1:91,2] = PR[GP1:90,2] + -37.019;
   1:L PR[91] R[100]mm/sec CNT100;
   1:  PR[GP1:91,1] = PR[GP1:90,1] + 34.246;
   1:  PR[GP1:91,2] = PR[GP1:90,2] + -35.615;
   1:L PR[91] R[100]mm/sec CNT100;
   1:  PR[GP1:91,1] = PR[GP1:90,1] + 41.844;
   1:  PR[GP1:91,2] = PR[GP1:90,2] + -26.463;
   1:L PR[91] R[100]mm/sec CNT100;
   1:  PR[GP1:91,1] = PR[GP1:90,1] + 42.743;
   1:  PR[GP1:91,2] = PR[GP1:90,2] + -24.697;
   1:L PR[91] R[100]mm/sec CNT100;
   1:  PR[GP1:91,1] = PR[GP1:90,1] + 47.545;
   1:  PR[GP1:91,2] = PR[GP1:90,2] + -13.821;
   1:L PR[91] R[100]mm/sec CNT100;
   1:  PR[GP1:91,1] = PR[GP1:90,1] + 49.190;
   1:  PR[GP1:91,2] = PR[GP1:90,2] + -2.023;
   1:L PR[91] R[100]mm/sec CNT100;
   1:  PR[GP1:91,1] = PR[GP1:90,1] + 49.500;
   1:  PR[GP1:91,2] = PR[GP1:90,2] + -0.066;
   1:L PR[91] R[100]mm/sec CNT100;
   1:  PR[GP1:91,1] = PR[GP1:90,1] + 47.857;
   1:  PR[GP1:91,2] = PR[GP1:90,2] + 11.715;
   1:L PR[91] R[100]mm/sec CNT100;
   1:  PR[GP1:91,1] = PR[GP1:90,1] + 47.547;
   1:  PR[GP1:91,2] = PR[GP1:90,2] + 13.672;
   1:L PR[91] R[100]mm/sec CNT100;
   1:  PR[GP1:91,1] = PR[GP1:90,1] + 42.743;
   1:  PR[GP1:91,2] = PR[GP1:90,2] + 24.553;
   1:L PR[91] R[100]mm/sec CNT100;
   1:  PR[GP1:91,1] = PR[GP1:90,1] + 41.844;
   1:  PR[GP1:91,2] = PR[GP1:90,2] + 26.319;
   1:L PR[91] R[100]mm/sec CNT100;
   1:  PR[GP1:91,1] = PR[GP1:90,1] + 34.246;
   1:  PR[GP1:91,2] = PR[GP1:90,2] + 35.471;
   1:L PR[91] R[100]mm/sec CNT100;
   1:  PR[GP1:91,1] = PR[GP1:90,1] + 32.842;
   1:  PR[GP1:91,2] = PR[GP1:90,2] + 36.875;
   1:L PR[91] R[100]mm/sec CNT100;
   1:  PR[GP1:91,1] = PR[GP1:90,1] + 24.212;
   1:  PR[GP1:91,2] = PR[GP1:90,2] + 42.986;
   1:L PR[91] R[100]mm/sec CNT100;
   1:  PR[GP1:91,1] = PR[GP1:90,1] + 22.438;
   1:  PR[GP1:91,2] = PR[GP1:90,2] + 43.890;
   1:L PR[91] R[100]mm/sec CNT100;
   1:  PR[GP1:91,1] = PR[GP1:90,1] + 12.577;
   1:  PR[GP1:91,2] = PR[GP1:90,2] + 47.711;
   1:L PR[91] R[100]mm/sec CNT100;
   1:  PR[GP1:91,1] = PR[GP1:90,1] + 10.611;
   1:  PR[GP1:91,2] = PR[GP1:90,2] + 48.022;
   1:L PR[91] R[100]mm/sec CNT100;
   1:  PR[GP1:91,1] = PR[GP1:90,1] + 0.105;
   1:  PR[GP1:91,2] = PR[GP1:90,2] + 49.323;
   1:L PR[91] R[100]mm/sec CNT100;
   1:  ! -- Layer/Ebene 213 -- !;
   1:  PR[91] = PR[90];
   1:  PR[GP1:91,1] = PR[GP1:90,1] + -9.656;
   1:  PR[GP1:91,2] = PR[GP1:90,2] + 48.114;
   1:  PR[GP1:91,3] = PR[GP1:90,3] + 130.235;
   1:L PR[91] R[100]mm/sec CNT100;
   1:  PR[GP1:91,1] = PR[GP1:90,1] + -12.564;
   1:  PR[GP1:91,2] = PR[GP1:90,2] + 47.653;
   1:L PR[91] R[100]mm/sec CNT100;
   1:  PR[GP1:91,1] = PR[GP1:90,1] + -21.724;
   1:  PR[GP1:91,2] = PR[GP1:90,2] + 44.104;
   1:L PR[91] R[100]mm/sec CNT100;
   1:  PR[GP1:91,1] = PR[GP1:90,1] + -24.348;
   1:  PR[GP1:91,2] = PR[GP1:90,2] + 42.767;
   1:L PR[91] R[100]mm/sec CNT100;
   1:  PR[GP1:91,1] = PR[GP1:90,1] + -32.365;
   1:  PR[GP1:91,2] = PR[GP1:90,2] + 37.090;
   1:L PR[91] R[100]mm/sec CNT100;
   1:  PR[GP1:91,1] = PR[GP1:90,1] + -34.446;
   1:  PR[GP1:91,2] = PR[GP1:90,2] + 35.009;
   1:L PR[91] R[100]mm/sec CNT100;
   1:  PR[GP1:91,1] = PR[GP1:90,1] + -41.504;
   1:  PR[GP1:91,2] = PR[GP1:90,2] + 26.507;
   1:L PR[91] R[100]mm/sec CNT100;
   1:  PR[GP1:91,1] = PR[GP1:90,1] + -42.837;
   1:  PR[GP1:91,2] = PR[GP1:90,2] + 23.891;
   1:L PR[91] R[100]mm/sec CNT100;
   1:  PR[GP1:91,1] = PR[GP1:90,1] + -47.298;
   1:  PR[GP1:91,2] = PR[GP1:90,2] + 13.785;
   1:L PR[91] R[100]mm/sec CNT100;
   1:  PR[GP1:91,1] = PR[GP1:90,1] + -48.828;
   1:  PR[GP1:91,2] = PR[GP1:90,2] + 2.821;
   1:L PR[91] R[100]mm/sec CNT100;
   1:  PR[GP1:91,1] = PR[GP1:90,1] + -49.287;
   1:  PR[GP1:91,2] = PR[GP1:90,2] + -0.078;
   1:L PR[91] R[100]mm/sec CNT100;
   1:  PR[GP1:91,1] = PR[GP1:90,1] + -47.760;
   1:  PR[GP1:91,2] = PR[GP1:90,2] + -11.025;
   1:L PR[91] R[100]mm/sec CNT100;
   1:  PR[GP1:91,1] = PR[GP1:90,1] + -47.301;
   1:  PR[GP1:91,2] = PR[GP1:90,2] + -13.924;
   1:L PR[91] R[100]mm/sec CNT100;
   1:  PR[GP1:91,1] = PR[GP1:90,1] + -42.837;
   1:  PR[GP1:91,2] = PR[GP1:90,2] + -24.035;
   1:L PR[91] R[100]mm/sec CNT100;
   1:  PR[GP1:91,1] = PR[GP1:90,1] + -41.504;
   1:  PR[GP1:91,2] = PR[GP1:90,2] + -26.651;
   1:L PR[91] R[100]mm/sec CNT100;
   1:  PR[GP1:91,1] = PR[GP1:90,1] + -34.446;
   1:  PR[GP1:91,2] = PR[GP1:90,2] + -35.153;
   1:L PR[91] R[100]mm/sec CNT100;
   1:  PR[GP1:91,1] = PR[GP1:90,1] + -32.365;
   1:  PR[GP1:91,2] = PR[GP1:90,2] + -37.234;
   1:L PR[91] R[100]mm/sec CNT100;
   1:  PR[GP1:91,1] = PR[GP1:90,1] + -24.348;
   1:  PR[GP1:91,2] = PR[GP1:90,2] + -42.911;
   1:L PR[91] R[100]mm/sec CNT100;
   1:  PR[GP1:91,1] = PR[GP1:90,1] + -21.724;
   1:  PR[GP1:91,2] = PR[GP1:90,2] + -44.248;
   1:L PR[91] R[100]mm/sec CNT100;
   1:  PR[GP1:91,1] = PR[GP1:90,1] + -12.574;
   1:  PR[GP1:91,2] = PR[GP1:90,2] + -47.794;
   1:L PR[91] R[100]mm/sec CNT100;
   1:  PR[GP1:91,1] = PR[GP1:90,1] + -2.793;
   1:  PR[GP1:91,2] = PR[GP1:90,2] + -49.005;
   1:L PR[91] R[100]mm/sec CNT100;
   1:  PR[GP1:91,1] = PR[GP1:90,1] + 0.115;
   1:  PR[GP1:91,2] = PR[GP1:90,2] + -49.466;
   1:L PR[91] R[100]mm/sec CNT100;
   1:  PR[GP1:91,1] = PR[GP1:90,1] + 9.867;
   1:  PR[GP1:91,2] = PR[GP1:90,2] + -48.259;
   1:L PR[91] R[100]mm/sec CNT100;
   1:  PR[GP1:91,1] = PR[GP1:90,1] + 12.776;
   1:  PR[GP1:91,2] = PR[GP1:90,2] + -47.798;
   1:L PR[91] R[100]mm/sec CNT100;
   1:  PR[GP1:91,1] = PR[GP1:90,1] + 21.937;
   1:  PR[GP1:91,2] = PR[GP1:90,2] + -44.248;
   1:L PR[91] R[100]mm/sec CNT100;
   1:  PR[GP1:91,1] = PR[GP1:90,1] + 24.561;
   1:  PR[GP1:91,2] = PR[GP1:90,2] + -42.911;
   1:L PR[91] R[100]mm/sec CNT100;
   1:  PR[GP1:91,1] = PR[GP1:90,1] + 32.580;
   1:  PR[GP1:91,2] = PR[GP1:90,2] + -37.232;
   1:L PR[91] R[100]mm/sec CNT100;
   1:  PR[GP1:91,1] = PR[GP1:90,1] + 34.658;
   1:  PR[GP1:91,2] = PR[GP1:90,2] + -35.154;
   1:L PR[91] R[100]mm/sec CNT100;
   1:  PR[GP1:91,1] = PR[GP1:90,1] + 41.718;
   1:  PR[GP1:91,2] = PR[GP1:90,2] + -26.650;
   1:L PR[91] R[100]mm/sec CNT100;
   1:  PR[GP1:91,1] = PR[GP1:90,1] + 43.051;
   1:  PR[GP1:91,2] = PR[GP1:90,2] + -24.035;
   1:L PR[91] R[100]mm/sec CNT100;
   1:  PR[GP1:91,1] = PR[GP1:90,1] + 47.512;
   1:  PR[GP1:91,2] = PR[GP1:90,2] + -13.929;
   1:L PR[91] R[100]mm/sec CNT100;
   1:  PR[GP1:91,1] = PR[GP1:90,1] + 49.041;
   1:  PR[GP1:91,2] = PR[GP1:90,2] + -2.965;
   1:L PR[91] R[100]mm/sec CNT100;
   1:  PR[GP1:91,1] = PR[GP1:90,1] + 49.500;
   1:  PR[GP1:91,2] = PR[GP1:90,2] + -0.066;
   1:L PR[91] R[100]mm/sec CNT100;
   1:  PR[GP1:91,1] = PR[GP1:90,1] + 47.973;
   1:  PR[GP1:91,2] = PR[GP1:90,2] + 10.881;
   1:L PR[91] R[100]mm/sec CNT100;
   1:  PR[GP1:91,1] = PR[GP1:90,1] + 47.514;
   1:  PR[GP1:91,2] = PR[GP1:90,2] + 13.780;
   1:L PR[91] R[100]mm/sec CNT100;
   1:  PR[GP1:91,1] = PR[GP1:90,1] + 43.051;
   1:  PR[GP1:91,2] = PR[GP1:90,2] + 23.891;
   1:L PR[91] R[100]mm/sec CNT100;
   1:  PR[GP1:91,1] = PR[GP1:90,1] + 41.718;
   1:  PR[GP1:91,2] = PR[GP1:90,2] + 26.506;
   1:L PR[91] R[100]mm/sec CNT100;
   1:  PR[GP1:91,1] = PR[GP1:90,1] + 34.659;
   1:  PR[GP1:91,2] = PR[GP1:90,2] + 35.010;
   1:L PR[91] R[100]mm/sec CNT100;
   1:  PR[GP1:91,1] = PR[GP1:90,1] + 32.580;
   1:  PR[GP1:91,2] = PR[GP1:90,2] + 37.089;
   1:L PR[91] R[100]mm/sec CNT100;
   1:  PR[GP1:91,1] = PR[GP1:90,1] + 24.561;
   1:  PR[GP1:91,2] = PR[GP1:90,2] + 42.767;
   1:L PR[91] R[100]mm/sec CNT100;
   1:  PR[GP1:91,1] = PR[GP1:90,1] + 21.937;
   1:  PR[GP1:91,2] = PR[GP1:90,2] + 44.104;
   1:L PR[91] R[100]mm/sec CNT100;
   1:  PR[GP1:91,1] = PR[GP1:90,1] + 12.776;
   1:  PR[GP1:91,2] = PR[GP1:90,2] + 47.654;
   1:L PR[91] R[100]mm/sec CNT100;
   1:  PR[GP1:91,1] = PR[GP1:90,1] + 9.867;
   1:  PR[GP1:91,2] = PR[GP1:90,2] + 48.115;
   1:L PR[91] R[100]mm/sec CNT100;
   1:  PR[GP1:91,1] = PR[GP1:90,1] + 0.105;
   1:  PR[GP1:91,2] = PR[GP1:90,2] + 49.323;
   1:L PR[91] R[100]mm/sec CNT100;
   1:  ! -- Layer/Ebene 214 -- !;
   1:  PR[91] = PR[90];
   1:  PR[GP1:91,1] = PR[GP1:90,1] + -8.911;
   1:  PR[GP1:91,2] = PR[GP1:90,2] + 48.206;
   1:  PR[GP1:91,3] = PR[GP1:90,3] + 130.845;
   1:L PR[91] R[100]mm/sec CNT100;
   1:  PR[GP1:91,1] = PR[GP1:90,1] + -12.762;
   1:  PR[GP1:91,2] = PR[GP1:90,2] + 47.596;
   1:L PR[91] R[100]mm/sec CNT100;
   1:  PR[GP1:91,1] = PR[GP1:90,1] + -21.223;
   1:  PR[GP1:91,2] = PR[GP1:90,2] + 44.317;
   1:L PR[91] R[100]mm/sec CNT100;
   1:  PR[GP1:91,1] = PR[GP1:90,1] + -24.698;
   1:  PR[GP1:91,2] = PR[GP1:90,2] + 42.547;
   1:L PR[91] R[100]mm/sec CNT100;
   1:  PR[GP1:91,1] = PR[GP1:90,1] + -32.103;
   1:  PR[GP1:91,2] = PR[GP1:90,2] + 37.304;
   1:L PR[91] R[100]mm/sec CNT100;
   1:  PR[GP1:91,1] = PR[GP1:90,1] + -34.858;
   1:  PR[GP1:91,2] = PR[GP1:90,2] + 34.549;
   1:L PR[91] R[100]mm/sec CNT100;
   1:  PR[GP1:91,1] = PR[GP1:90,1] + -41.378;
   1:  PR[GP1:91,2] = PR[GP1:90,2] + 26.694;
   1:L PR[91] R[100]mm/sec CNT100;
   1:  PR[GP1:91,1] = PR[GP1:90,1] + -43.144;
   1:  PR[GP1:91,2] = PR[GP1:90,2] + 23.228;
   1:L PR[91] R[100]mm/sec CNT100;
   1:  PR[GP1:91,1] = PR[GP1:90,1] + -47.266;
   1:  PR[GP1:91,2] = PR[GP1:90,2] + 13.893;
   1:L PR[91] R[100]mm/sec CNT100;
   1:  PR[GP1:91,1] = PR[GP1:90,1] + -48.678;
   1:  PR[GP1:91,2] = PR[GP1:90,2] + 3.764;
   1:L PR[91] R[100]mm/sec CNT100;
   1:  PR[GP1:91,1] = PR[GP1:90,1] + -49.287;
   1:  PR[GP1:91,2] = PR[GP1:90,2] + -0.078;
   1:L PR[91] R[100]mm/sec CNT100;
   1:  PR[GP1:91,1] = PR[GP1:90,1] + -47.876;
   1:  PR[GP1:91,2] = PR[GP1:90,2] + -10.191;
   1:L PR[91] R[100]mm/sec CNT100;
   1:  PR[GP1:91,1] = PR[GP1:90,1] + -47.268;
   1:  PR[GP1:91,2] = PR[GP1:90,2] + -14.032;
   1:L PR[91] R[100]mm/sec CNT100;
   1:  PR[GP1:91,1] = PR[GP1:90,1] + -43.144;
   1:  PR[GP1:91,2] = PR[GP1:90,2] + -23.372;
   1:L PR[91] R[100]mm/sec CNT100;
   1:  PR[GP1:91,1] = PR[GP1:90,1] + -41.378;
   1:  PR[GP1:91,2] = PR[GP1:90,2] + -26.838;
   1:L PR[91] R[100]mm/sec CNT100;
   1:  PR[GP1:91,1] = PR[GP1:90,1] + -34.858;
   1:  PR[GP1:91,2] = PR[GP1:90,2] + -34.693;
   1:L PR[91] R[100]mm/sec CNT100;
   1:  PR[GP1:91,1] = PR[GP1:90,1] + -32.103;
   1:  PR[GP1:91,2] = PR[GP1:90,2] + -37.448;
   1:L PR[91] R[100]mm/sec CNT100;
   1:  PR[GP1:91,1] = PR[GP1:90,1] + -24.698;
   1:  PR[GP1:91,2] = PR[GP1:90,2] + -42.691;
   1:L PR[91] R[100]mm/sec CNT100;
   1:  PR[GP1:91,1] = PR[GP1:90,1] + -21.223;
   1:  PR[GP1:91,2] = PR[GP1:90,2] + -44.461;
   1:L PR[91] R[100]mm/sec CNT100;
   1:  PR[GP1:91,1] = PR[GP1:90,1] + -12.772;
   1:  PR[GP1:91,2] = PR[GP1:90,2] + -47.737;
   1:L PR[91] R[100]mm/sec CNT100;
   1:  PR[GP1:91,1] = PR[GP1:90,1] + -3.736;
   1:  PR[GP1:91,2] = PR[GP1:90,2] + -48.856;
   1:L PR[91] R[100]mm/sec CNT100;
   1:  PR[GP1:91,1] = PR[GP1:90,1] + 0.115;
   1:  PR[GP1:91,2] = PR[GP1:90,2] + -49.466;
   1:L PR[91] R[100]mm/sec CNT100;
   1:  PR[GP1:91,1] = PR[GP1:90,1] + 9.123;
   1:  PR[GP1:91,2] = PR[GP1:90,2] + -48.351;
   1:L PR[91] R[100]mm/sec CNT100;
   1:  PR[GP1:91,1] = PR[GP1:90,1] + 12.974;
   1:  PR[GP1:91,2] = PR[GP1:90,2] + -47.741;
   1:L PR[91] R[100]mm/sec CNT100;
   1:  PR[GP1:91,1] = PR[GP1:90,1] + 21.436;
   1:  PR[GP1:91,2] = PR[GP1:90,2] + -44.462;
   1:L PR[91] R[100]mm/sec CNT100;
   1:  PR[GP1:91,1] = PR[GP1:90,1] + 24.911;
   1:  PR[GP1:91,2] = PR[GP1:90,2] + -42.691;
   1:L PR[91] R[100]mm/sec CNT100;
   1:  PR[GP1:91,1] = PR[GP1:90,1] + 32.317;
   1:  PR[GP1:91,2] = PR[GP1:90,2] + -37.446;
   1:L PR[91] R[100]mm/sec CNT100;
   1:  PR[GP1:91,1] = PR[GP1:90,1] + 35.071;
   1:  PR[GP1:91,2] = PR[GP1:90,2] + -34.693;
   1:L PR[91] R[100]mm/sec CNT100;
   1:  PR[GP1:91,1] = PR[GP1:90,1] + 41.592;
   1:  PR[GP1:91,2] = PR[GP1:90,2] + -26.837;
   1:L PR[91] R[100]mm/sec CNT100;
   1:  PR[GP1:91,1] = PR[GP1:90,1] + 43.358;
   1:  PR[GP1:91,2] = PR[GP1:90,2] + -23.372;
   1:L PR[91] R[100]mm/sec CNT100;
   1:  PR[GP1:91,1] = PR[GP1:90,1] + 47.479;
   1:  PR[GP1:91,2] = PR[GP1:90,2] + -14.037;
   1:L PR[91] R[100]mm/sec CNT100;
   1:  PR[GP1:91,1] = PR[GP1:90,1] + 48.892;
   1:  PR[GP1:91,2] = PR[GP1:90,2] + -3.908;
   1:L PR[91] R[100]mm/sec CNT100;
   1:  PR[GP1:91,1] = PR[GP1:90,1] + 49.500;
   1:  PR[GP1:91,2] = PR[GP1:90,2] + -0.066;
   1:L PR[91] R[100]mm/sec CNT100;
   1:  PR[GP1:91,1] = PR[GP1:90,1] + 48.090;
   1:  PR[GP1:91,2] = PR[GP1:90,2] + 10.046;
   1:L PR[91] R[100]mm/sec CNT100;
   1:  PR[GP1:91,1] = PR[GP1:90,1] + 47.481;
   1:  PR[GP1:91,2] = PR[GP1:90,2] + 13.888;
   1:L PR[91] R[100]mm/sec CNT100;
   1:  PR[GP1:91,1] = PR[GP1:90,1] + 43.358;
   1:  PR[GP1:91,2] = PR[GP1:90,2] + 23.228;
   1:L PR[91] R[100]mm/sec CNT100;
   1:  PR[GP1:91,1] = PR[GP1:90,1] + 41.592;
   1:  PR[GP1:91,2] = PR[GP1:90,2] + 26.693;
   1:L PR[91] R[100]mm/sec CNT100;
   1:  PR[GP1:91,1] = PR[GP1:90,1] + 35.071;
   1:  PR[GP1:91,2] = PR[GP1:90,2] + 34.549;
   1:L PR[91] R[100]mm/sec CNT100;
   1:  PR[GP1:91,1] = PR[GP1:90,1] + 32.317;
   1:  PR[GP1:91,2] = PR[GP1:90,2] + 37.302;
   1:L PR[91] R[100]mm/sec CNT100;
   1:  PR[GP1:91,1] = PR[GP1:90,1] + 24.911;
   1:  PR[GP1:91,2] = PR[GP1:90,2] + 42.547;
   1:L PR[91] R[100]mm/sec CNT100;
   1:  PR[GP1:91,1] = PR[GP1:90,1] + 21.436;
   1:  PR[GP1:91,2] = PR[GP1:90,2] + 44.318;
   1:L PR[91] R[100]mm/sec CNT100;
   1:  PR[GP1:91,1] = PR[GP1:90,1] + 12.974;
   1:  PR[GP1:91,2] = PR[GP1:90,2] + 47.597;
   1:L PR[91] R[100]mm/sec CNT100;
   1:  PR[GP1:91,1] = PR[GP1:90,1] + 9.123;
   1:  PR[GP1:91,2] = PR[GP1:90,2] + 48.207;
   1:L PR[91] R[100]mm/sec CNT100;
   1:  PR[GP1:91,1] = PR[GP1:90,1] + 0.105;
   1:  PR[GP1:91,2] = PR[GP1:90,2] + 49.323;
   1:L PR[91] R[100]mm/sec CNT100;
   1:  ! -- Layer/Ebene 215 -- !;
   1:  PR[91] = PR[90];
   1:  PR[GP1:91,1] = PR[GP1:90,1] + -8.167;
   1:  PR[GP1:91,2] = PR[GP1:90,2] + 48.298;
   1:  PR[GP1:91,3] = PR[GP1:90,3] + 131.455;
   1:L PR[91] R[100]mm/sec CNT100;
   1:  PR[GP1:91,1] = PR[GP1:90,1] + -12.961;
   1:  PR[GP1:91,2] = PR[GP1:90,2] + 47.539;
   1:L PR[91] R[100]mm/sec CNT100;
   1:  PR[GP1:91,1] = PR[GP1:90,1] + -20.722;
   1:  PR[GP1:91,2] = PR[GP1:90,2] + 44.531;
   1:L PR[91] R[100]mm/sec CNT100;
   1:  PR[GP1:91,1] = PR[GP1:90,1] + -25.047;
   1:  PR[GP1:91,2] = PR[GP1:90,2] + 42.328;
   1:L PR[91] R[100]mm/sec CNT100;
   1:  PR[GP1:91,1] = PR[GP1:90,1] + -31.840;
   1:  PR[GP1:91,2] = PR[GP1:90,2] + 37.518;
   1:L PR[91] R[100]mm/sec CNT100;
   1:  PR[GP1:91,1] = PR[GP1:90,1] + -35.270;
   1:  PR[GP1:91,2] = PR[GP1:90,2] + 34.088;
   1:L PR[91] R[100]mm/sec CNT100;
   1:  PR[GP1:91,1] = PR[GP1:90,1] + -41.253;
   1:  PR[GP1:91,2] = PR[GP1:90,2] + 26.881;
   1:L PR[91] R[100]mm/sec CNT100;
   1:  PR[GP1:91,1] = PR[GP1:90,1] + -43.452;
   1:  PR[GP1:91,2] = PR[GP1:90,2] + 22.565;
   1:L PR[91] R[100]mm/sec CNT100;
   1:  PR[GP1:91,1] = PR[GP1:90,1] + -47.233;
   1:  PR[GP1:91,2] = PR[GP1:90,2] + 14.001;
   1:L PR[91] R[100]mm/sec CNT100;
   1:  PR[GP1:91,1] = PR[GP1:90,1] + -48.529;
   1:  PR[GP1:91,2] = PR[GP1:90,2] + 4.706;
   1:L PR[91] R[100]mm/sec CNT100;
   1:  PR[GP1:91,1] = PR[GP1:90,1] + -49.287;
   1:  PR[GP1:91,2] = PR[GP1:90,2] + -0.078;
   1:L PR[91] R[100]mm/sec CNT100;
   1:  PR[GP1:91,1] = PR[GP1:90,1] + -47.993;
   1:  PR[GP1:91,2] = PR[GP1:90,2] + -9.356;
   1:L PR[91] R[100]mm/sec CNT100;
   1:  PR[GP1:91,1] = PR[GP1:90,1] + -47.235;
   1:  PR[GP1:91,2] = PR[GP1:90,2] + -14.140;
   1:L PR[91] R[100]mm/sec CNT100;
   1:  PR[GP1:91,1] = PR[GP1:90,1] + -43.452;
   1:  PR[GP1:91,2] = PR[GP1:90,2] + -22.709;
   1:L PR[91] R[100]mm/sec CNT100;
   1:  PR[GP1:91,1] = PR[GP1:90,1] + -41.253;
   1:  PR[GP1:91,2] = PR[GP1:90,2] + -27.025;
   1:L PR[91] R[100]mm/sec CNT100;
   1:  PR[GP1:91,1] = PR[GP1:90,1] + -35.270;
   1:  PR[GP1:91,2] = PR[GP1:90,2] + -34.232;
   1:L PR[91] R[100]mm/sec CNT100;
   1:  PR[GP1:91,1] = PR[GP1:90,1] + -31.840;
   1:  PR[GP1:91,2] = PR[GP1:90,2] + -37.661;
   1:L PR[91] R[100]mm/sec CNT100;
   1:  PR[GP1:91,1] = PR[GP1:90,1] + -25.047;
   1:  PR[GP1:91,2] = PR[GP1:90,2] + -42.472;
   1:L PR[91] R[100]mm/sec CNT100;
   1:  PR[GP1:91,1] = PR[GP1:90,1] + -20.722;
   1:  PR[GP1:91,2] = PR[GP1:90,2] + -44.675;
   1:L PR[91] R[100]mm/sec CNT100;
   1:  PR[GP1:91,1] = PR[GP1:90,1] + -12.970;
   1:  PR[GP1:91,2] = PR[GP1:90,2] + -47.679;
   1:L PR[91] R[100]mm/sec CNT100;
   1:  PR[GP1:91,1] = PR[GP1:90,1] + -4.678;
   1:  PR[GP1:91,2] = PR[GP1:90,2] + -48.707;
   1:L PR[91] R[100]mm/sec CNT100;
   1:  PR[GP1:91,1] = PR[GP1:90,1] + 0.115;
   1:  PR[GP1:91,2] = PR[GP1:90,2] + -49.466;
   1:L PR[91] R[100]mm/sec CNT100;
   1:  PR[GP1:91,1] = PR[GP1:90,1] + 8.379;
   1:  PR[GP1:91,2] = PR[GP1:90,2] + -48.443;
   1:L PR[91] R[100]mm/sec CNT100;
   1:  PR[GP1:91,1] = PR[GP1:90,1] + 13.173;
   1:  PR[GP1:91,2] = PR[GP1:90,2] + -47.684;
   1:L PR[91] R[100]mm/sec CNT100;
   1:  PR[GP1:91,1] = PR[GP1:90,1] + 20.935;
   1:  PR[GP1:91,2] = PR[GP1:90,2] + -44.675;
   1:L PR[91] R[100]mm/sec CNT100;
   1:  PR[GP1:91,1] = PR[GP1:90,1] + 25.260;
   1:  PR[GP1:91,2] = PR[GP1:90,2] + -42.472;
   1:L PR[91] R[100]mm/sec CNT100;
   1:  PR[GP1:91,1] = PR[GP1:90,1] + 32.055;
   1:  PR[GP1:91,2] = PR[GP1:90,2] + -37.660;
   1:L PR[91] R[100]mm/sec CNT100;
   1:  PR[GP1:91,1] = PR[GP1:90,1] + 35.483;
   1:  PR[GP1:91,2] = PR[GP1:90,2] + -34.232;
   1:L PR[91] R[100]mm/sec CNT100;
   1:  PR[GP1:91,1] = PR[GP1:90,1] + 41.466;
   1:  PR[GP1:91,2] = PR[GP1:90,2] + -27.025;
   1:L PR[91] R[100]mm/sec CNT100;
   1:  PR[GP1:91,1] = PR[GP1:90,1] + 43.665;
   1:  PR[GP1:91,2] = PR[GP1:90,2] + -22.709;
   1:L PR[91] R[100]mm/sec CNT100;
   1:  PR[GP1:91,1] = PR[GP1:90,1] + 47.446;
   1:  PR[GP1:91,2] = PR[GP1:90,2] + -14.145;
   1:L PR[91] R[100]mm/sec CNT100;
   1:  PR[GP1:91,1] = PR[GP1:90,1] + 48.742;
   1:  PR[GP1:91,2] = PR[GP1:90,2] + -4.850;
   1:L PR[91] R[100]mm/sec CNT100;
   1:  PR[GP1:91,1] = PR[GP1:90,1] + 49.500;
   1:  PR[GP1:91,2] = PR[GP1:90,2] + -0.066;
   1:L PR[91] R[100]mm/sec CNT100;
   1:  PR[GP1:91,1] = PR[GP1:90,1] + 48.206;
   1:  PR[GP1:91,2] = PR[GP1:90,2] + 9.212;
   1:L PR[91] R[100]mm/sec CNT100;
   1:  PR[GP1:91,1] = PR[GP1:90,1] + 47.448;
   1:  PR[GP1:91,2] = PR[GP1:90,2] + 13.996;
   1:L PR[91] R[100]mm/sec CNT100;
   1:  PR[GP1:91,1] = PR[GP1:90,1] + 43.665;
   1:  PR[GP1:91,2] = PR[GP1:90,2] + 22.565;
   1:L PR[91] R[100]mm/sec CNT100;
   1:  PR[GP1:91,1] = PR[GP1:90,1] + 41.466;
   1:  PR[GP1:91,2] = PR[GP1:90,2] + 26.881;
   1:L PR[91] R[100]mm/sec CNT100;
   1:  PR[GP1:91,1] = PR[GP1:90,1] + 35.483;
   1:  PR[GP1:91,2] = PR[GP1:90,2] + 34.088;
   1:L PR[91] R[100]mm/sec CNT100;
   1:  PR[GP1:91,1] = PR[GP1:90,1] + 32.055;
   1:  PR[GP1:91,2] = PR[GP1:90,2] + 37.516;
   1:L PR[91] R[100]mm/sec CNT100;
   1:  PR[GP1:91,1] = PR[GP1:90,1] + 25.260;
   1:  PR[GP1:91,2] = PR[GP1:90,2] + 42.328;
   1:L PR[91] R[100]mm/sec CNT100;
   1:  PR[GP1:91,1] = PR[GP1:90,1] + 20.935;
   1:  PR[GP1:91,2] = PR[GP1:90,2] + 44.531;
   1:L PR[91] R[100]mm/sec CNT100;
   1:  PR[GP1:91,1] = PR[GP1:90,1] + 13.173;
   1:  PR[GP1:91,2] = PR[GP1:90,2] + 47.540;
   1:L PR[91] R[100]mm/sec CNT100;
   1:  PR[GP1:91,1] = PR[GP1:90,1] + 8.379;
   1:  PR[GP1:91,2] = PR[GP1:90,2] + 48.299;
   1:L PR[91] R[100]mm/sec CNT100;
   1:  PR[GP1:91,1] = PR[GP1:90,1] + 0.105;
   1:  PR[GP1:91,2] = PR[GP1:90,2] + 49.323;
   1:L PR[91] R[100]mm/sec CNT100;
   1:  ! -- Layer/Ebene 216 -- !;
   1:  PR[91] = PR[90];
   1:  PR[GP1:91,1] = PR[GP1:90,1] + -7.423;
   1:  PR[GP1:91,2] = PR[GP1:90,2] + 48.391;
   1:  PR[GP1:91,3] = PR[GP1:90,3] + 132.065;
   1:L PR[91] R[100]mm/sec CNT100;
   1:  PR[GP1:91,1] = PR[GP1:90,1] + -13.159;
   1:  PR[GP1:91,2] = PR[GP1:90,2] + 47.482;
   1:L PR[91] R[100]mm/sec CNT100;
   1:  PR[GP1:91,1] = PR[GP1:90,1] + -20.222;
   1:  PR[GP1:91,2] = PR[GP1:90,2] + 44.745;
   1:L PR[91] R[100]mm/sec CNT100;
   1:  PR[GP1:91,1] = PR[GP1:90,1] + -25.396;
   1:  PR[GP1:91,2] = PR[GP1:90,2] + 42.108;
   1:L PR[91] R[100]mm/sec CNT100;
   1:  PR[GP1:91,1] = PR[GP1:90,1] + -31.578;
   1:  PR[GP1:91,2] = PR[GP1:90,2] + 37.731;
   1:L PR[91] R[100]mm/sec CNT100;
   1:  PR[GP1:91,1] = PR[GP1:90,1] + -35.682;
   1:  PR[GP1:91,2] = PR[GP1:90,2] + 33.627;
   1:L PR[91] R[100]mm/sec CNT100;
   1:  PR[GP1:91,1] = PR[GP1:90,1] + -41.127;
   1:  PR[GP1:91,2] = PR[GP1:90,2] + 27.069;
   1:L PR[91] R[100]mm/sec CNT100;
   1:  PR[GP1:91,1] = PR[GP1:90,1] + -43.759;
   1:  PR[GP1:91,2] = PR[GP1:90,2] + 21.902;
   1:L PR[91] R[100]mm/sec CNT100;
   1:  PR[GP1:91,1] = PR[GP1:90,1] + -47.200;
   1:  PR[GP1:91,2] = PR[GP1:90,2] + 14.109;
   1:L PR[91] R[100]mm/sec CNT100;
   1:  PR[GP1:91,1] = PR[GP1:90,1] + -48.380;
   1:  PR[GP1:91,2] = PR[GP1:90,2] + 5.649;
   1:L PR[91] R[100]mm/sec CNT100;
   1:  PR[GP1:91,1] = PR[GP1:90,1] + -49.287;
   1:  PR[GP1:91,2] = PR[GP1:90,2] + -0.078;
   1:L PR[91] R[100]mm/sec CNT100;
   1:  PR[GP1:91,1] = PR[GP1:90,1] + -48.109;
   1:  PR[GP1:91,2] = PR[GP1:90,2] + -8.521;
   1:L PR[91] R[100]mm/sec CNT100;
   1:  PR[GP1:91,1] = PR[GP1:90,1] + -47.202;
   1:  PR[GP1:91,2] = PR[GP1:90,2] + -14.248;
   1:L PR[91] R[100]mm/sec CNT100;
   1:  PR[GP1:91,1] = PR[GP1:90,1] + -43.759;
   1:  PR[GP1:91,2] = PR[GP1:90,2] + -22.046;
   1:L PR[91] R[100]mm/sec CNT100;
   1:  PR[GP1:91,1] = PR[GP1:90,1] + -41.127;
   1:  PR[GP1:91,2] = PR[GP1:90,2] + -27.213;
   1:L PR[91] R[100]mm/sec CNT100;
   1:  PR[GP1:91,1] = PR[GP1:90,1] + -35.683;
   1:  PR[GP1:91,2] = PR[GP1:90,2] + -33.771;
   1:L PR[91] R[100]mm/sec CNT100;
   1:  PR[GP1:91,1] = PR[GP1:90,1] + -31.578;
   1:  PR[GP1:91,2] = PR[GP1:90,2] + -37.875;
   1:L PR[91] R[100]mm/sec CNT100;
   1:  PR[GP1:91,1] = PR[GP1:90,1] + -25.397;
   1:  PR[GP1:91,2] = PR[GP1:90,2] + -42.252;
   1:L PR[91] R[100]mm/sec CNT100;
   1:  PR[GP1:91,1] = PR[GP1:90,1] + -20.222;
   1:  PR[GP1:91,2] = PR[GP1:90,2] + -44.889;
   1:L PR[91] R[100]mm/sec CNT100;
   1:  PR[GP1:91,1] = PR[GP1:90,1] + -13.169;
   1:  PR[GP1:91,2] = PR[GP1:90,2] + -47.622;
   1:L PR[91] R[100]mm/sec CNT100;
   1:  PR[GP1:91,1] = PR[GP1:90,1] + -5.620;
   1:  PR[GP1:91,2] = PR[GP1:90,2] + -48.558;
   1:L PR[91] R[100]mm/sec CNT100;
   1:  PR[GP1:91,1] = PR[GP1:90,1] + 0.116;
   1:  PR[GP1:91,2] = PR[GP1:90,2] + -49.466;
   1:L PR[91] R[100]mm/sec CNT100;
   1:  PR[GP1:91,1] = PR[GP1:90,1] + 7.635;
   1:  PR[GP1:91,2] = PR[GP1:90,2] + -48.535;
   1:L PR[91] R[100]mm/sec CNT100;
   1:  PR[GP1:91,1] = PR[GP1:90,1] + 13.371;
   1:  PR[GP1:91,2] = PR[GP1:90,2] + -47.626;
   1:L PR[91] R[100]mm/sec CNT100;
   1:  PR[GP1:91,1] = PR[GP1:90,1] + 20.435;
   1:  PR[GP1:91,2] = PR[GP1:90,2] + -44.889;
   1:L PR[91] R[100]mm/sec CNT100;
   1:  PR[GP1:91,1] = PR[GP1:90,1] + 25.610;
   1:  PR[GP1:91,2] = PR[GP1:90,2] + -42.252;
   1:L PR[91] R[100]mm/sec CNT100;
   1:  PR[GP1:91,1] = PR[GP1:90,1] + 31.792;
   1:  PR[GP1:91,2] = PR[GP1:90,2] + -37.874;
   1:L PR[91] R[100]mm/sec CNT100;
   1:  PR[GP1:91,1] = PR[GP1:90,1] + 35.896;
   1:  PR[GP1:91,2] = PR[GP1:90,2] + -33.771;
   1:L PR[91] R[100]mm/sec CNT100;
   1:  PR[GP1:91,1] = PR[GP1:90,1] + 41.340;
   1:  PR[GP1:91,2] = PR[GP1:90,2] + -27.212;
   1:L PR[91] R[100]mm/sec CNT100;
   1:  PR[GP1:91,1] = PR[GP1:90,1] + 43.973;
   1:  PR[GP1:91,2] = PR[GP1:90,2] + -22.046;
   1:L PR[91] R[100]mm/sec CNT100;
   1:  PR[GP1:91,1] = PR[GP1:90,1] + 47.413;
   1:  PR[GP1:91,2] = PR[GP1:90,2] + -14.253;
   1:L PR[91] R[100]mm/sec CNT100;
   1:  PR[GP1:91,1] = PR[GP1:90,1] + 48.593;
   1:  PR[GP1:91,2] = PR[GP1:90,2] + -5.793;
   1:L PR[91] R[100]mm/sec CNT100;
   1:  PR[GP1:91,1] = PR[GP1:90,1] + 49.500;
   1:  PR[GP1:91,2] = PR[GP1:90,2] + -0.066;
   1:L PR[91] R[100]mm/sec CNT100;
   1:  PR[GP1:91,1] = PR[GP1:90,1] + 48.322;
   1:  PR[GP1:91,2] = PR[GP1:90,2] + 8.377;
   1:L PR[91] R[100]mm/sec CNT100;
   1:  PR[GP1:91,1] = PR[GP1:90,1] + 47.415;
   1:  PR[GP1:91,2] = PR[GP1:90,2] + 14.104;
   1:L PR[91] R[100]mm/sec CNT100;
   1:  PR[GP1:91,1] = PR[GP1:90,1] + 43.973;
   1:  PR[GP1:91,2] = PR[GP1:90,2] + 21.902;
   1:L PR[91] R[100]mm/sec CNT100;
   1:  PR[GP1:91,1] = PR[GP1:90,1] + 41.340;
   1:  PR[GP1:91,2] = PR[GP1:90,2] + 27.068;
   1:L PR[91] R[100]mm/sec CNT100;
   1:  PR[GP1:91,1] = PR[GP1:90,1] + 35.895;
   1:  PR[GP1:91,2] = PR[GP1:90,2] + 33.627;
   1:L PR[91] R[100]mm/sec CNT100;
   1:  PR[GP1:91,1] = PR[GP1:90,1] + 31.792;
   1:  PR[GP1:91,2] = PR[GP1:90,2] + 37.730;
   1:L PR[91] R[100]mm/sec CNT100;
   1:  PR[GP1:91,1] = PR[GP1:90,1] + 25.610;
   1:  PR[GP1:91,2] = PR[GP1:90,2] + 42.109;
   1:L PR[91] R[100]mm/sec CNT100;
   1:  PR[GP1:91,1] = PR[GP1:90,1] + 20.435;
   1:  PR[GP1:91,2] = PR[GP1:90,2] + 44.745;
   1:L PR[91] R[100]mm/sec CNT100;
   1:  PR[GP1:91,1] = PR[GP1:90,1] + 13.371;
   1:  PR[GP1:91,2] = PR[GP1:90,2] + 47.482;
   1:L PR[91] R[100]mm/sec CNT100;
   1:  PR[GP1:91,1] = PR[GP1:90,1] + 7.635;
   1:  PR[GP1:91,2] = PR[GP1:90,2] + 48.391;
   1:L PR[91] R[100]mm/sec CNT100;
   1:  PR[GP1:91,1] = PR[GP1:90,1] + 0.105;
   1:  PR[GP1:91,2] = PR[GP1:90,2] + 49.323;
   1:L PR[91] R[100]mm/sec CNT100;
   1:  ! -- Layer/Ebene 217 -- !;
   1:  PR[91] = PR[90];
   1:  PR[GP1:91,1] = PR[GP1:90,1] + -6.679;
   1:  PR[GP1:91,2] = PR[GP1:90,2] + 48.483;
   1:  PR[GP1:91,3] = PR[GP1:90,3] + 132.675;
   1:L PR[91] R[100]mm/sec CNT100;
   1:  PR[GP1:91,1] = PR[GP1:90,1] + -13.357;
   1:  PR[GP1:91,2] = PR[GP1:90,2] + 47.425;
   1:L PR[91] R[100]mm/sec CNT100;
   1:  PR[GP1:91,1] = PR[GP1:90,1] + -19.721;
   1:  PR[GP1:91,2] = PR[GP1:90,2] + 44.959;
   1:L PR[91] R[100]mm/sec CNT100;
   1:  PR[GP1:91,1] = PR[GP1:90,1] + -25.746;
   1:  PR[GP1:91,2] = PR[GP1:90,2] + 41.889;
   1:L PR[91] R[100]mm/sec CNT100;
   1:  PR[GP1:91,1] = PR[GP1:90,1] + -31.316;
   1:  PR[GP1:91,2] = PR[GP1:90,2] + 37.945;
   1:L PR[91] R[100]mm/sec CNT100;
   1:  PR[GP1:91,1] = PR[GP1:90,1] + -36.095;
   1:  PR[GP1:91,2] = PR[GP1:90,2] + 33.166;
   1:L PR[91] R[100]mm/sec CNT100;
   1:  PR[GP1:91,1] = PR[GP1:90,1] + -41.001;
   1:  PR[GP1:91,2] = PR[GP1:90,2] + 27.256;
   1:L PR[91] R[100]mm/sec CNT100;
   1:  PR[GP1:91,1] = PR[GP1:90,1] + -44.067;
   1:  PR[GP1:91,2] = PR[GP1:90,2] + 21.240;
   1:L PR[91] R[100]mm/sec CNT100;
   1:  PR[GP1:91,1] = PR[GP1:90,1] + -47.167;
   1:  PR[GP1:91,2] = PR[GP1:90,2] + 14.217;
   1:L PR[91] R[100]mm/sec CNT100;
   1:  PR[GP1:91,1] = PR[GP1:90,1] + -48.230;
   1:  PR[GP1:91,2] = PR[GP1:90,2] + 6.591;
   1:L PR[91] R[100]mm/sec CNT100;
   1:  PR[GP1:91,1] = PR[GP1:90,1] + -49.287;
   1:  PR[GP1:91,2] = PR[GP1:90,2] + -0.078;
   1:L PR[91] R[100]mm/sec CNT100;
   1:  PR[GP1:91,1] = PR[GP1:90,1] + -48.225;
   1:  PR[GP1:91,2] = PR[GP1:90,2] + -7.687;
   1:L PR[91] R[100]mm/sec CNT100;
   1:  PR[GP1:91,1] = PR[GP1:90,1] + -47.169;
   1:  PR[GP1:91,2] = PR[GP1:90,2] + -14.356;
   1:L PR[91] R[100]mm/sec CNT100;
   1:  PR[GP1:91,1] = PR[GP1:90,1] + -44.067;
   1:  PR[GP1:91,2] = PR[GP1:90,2] + -21.384;
   1:L PR[91] R[100]mm/sec CNT100;
   1:  PR[GP1:91,1] = PR[GP1:90,1] + -41.001;
   1:  PR[GP1:91,2] = PR[GP1:90,2] + -27.400;
   1:L PR[91] R[100]mm/sec CNT100;
   1:  PR[GP1:91,1] = PR[GP1:90,1] + -36.095;
   1:  PR[GP1:91,2] = PR[GP1:90,2] + -33.310;
   1:L PR[91] R[100]mm/sec CNT100;
   1:  PR[GP1:91,1] = PR[GP1:90,1] + -31.316;
   1:  PR[GP1:91,2] = PR[GP1:90,2] + -38.089;
   1:L PR[91] R[100]mm/sec CNT100;
   1:  PR[GP1:91,1] = PR[GP1:90,1] + -25.746;
   1:  PR[GP1:91,2] = PR[GP1:90,2] + -42.033;
   1:L PR[91] R[100]mm/sec CNT100;
   1:  PR[GP1:91,1] = PR[GP1:90,1] + -19.721;
   1:  PR[GP1:91,2] = PR[GP1:90,2] + -45.103;
   1:L PR[91] R[100]mm/sec CNT100;
   1:  PR[GP1:91,1] = PR[GP1:90,1] + -13.367;
   1:  PR[GP1:91,2] = PR[GP1:90,2] + -47.565;
   1:L PR[91] R[100]mm/sec CNT100;
   1:  PR[GP1:91,1] = PR[GP1:90,1] + -6.563;
   1:  PR[GP1:91,2] = PR[GP1:90,2] + -48.408;
   1:L PR[91] R[100]mm/sec CNT100;
   1:  PR[GP1:91,1] = PR[GP1:90,1] + 0.116;
   1:  PR[GP1:91,2] = PR[GP1:90,2] + -49.466;
   1:L PR[91] R[100]mm/sec CNT100;
   1:  PR[GP1:91,1] = PR[GP1:90,1] + 6.891;
   1:  PR[GP1:91,2] = PR[GP1:90,2] + -48.627;
   1:L PR[91] R[100]mm/sec CNT100;
   1:  PR[GP1:91,1] = PR[GP1:90,1] + 13.569;
   1:  PR[GP1:91,2] = PR[GP1:90,2] + -47.569;
   1:L PR[91] R[100]mm/sec CNT100;
   1:  PR[GP1:91,1] = PR[GP1:90,1] + 19.934;
   1:  PR[GP1:91,2] = PR[GP1:90,2] + -45.103;
   1:L PR[91] R[100]mm/sec CNT100;
   1:  PR[GP1:91,1] = PR[GP1:90,1] + 25.959;
   1:  PR[GP1:91,2] = PR[GP1:90,2] + -42.033;
   1:L PR[91] R[100]mm/sec CNT100;
   1:  PR[GP1:91,1] = PR[GP1:90,1] + 31.530;
   1:  PR[GP1:91,2] = PR[GP1:90,2] + -38.088;
   1:L PR[91] R[100]mm/sec CNT100;
   1:  PR[GP1:91,1] = PR[GP1:90,1] + 36.308;
   1:  PR[GP1:91,2] = PR[GP1:90,2] + -33.310;
   1:L PR[91] R[100]mm/sec CNT100;
   1:  PR[GP1:91,1] = PR[GP1:90,1] + 41.215;
   1:  PR[GP1:91,2] = PR[GP1:90,2] + -27.400;
   1:L PR[91] R[100]mm/sec CNT100;
   1:  PR[GP1:91,1] = PR[GP1:90,1] + 44.280;
   1:  PR[GP1:91,2] = PR[GP1:90,2] + -21.383;
   1:L PR[91] R[100]mm/sec CNT100;
   1:  PR[GP1:91,1] = PR[GP1:90,1] + 47.380;
   1:  PR[GP1:91,2] = PR[GP1:90,2] + -14.361;
   1:L PR[91] R[100]mm/sec CNT100;
   1:  PR[GP1:91,1] = PR[GP1:90,1] + 48.444;
   1:  PR[GP1:91,2] = PR[GP1:90,2] + -6.735;
   1:L PR[91] R[100]mm/sec CNT100;
   1:  PR[GP1:91,1] = PR[GP1:90,1] + 49.500;
   1:  PR[GP1:91,2] = PR[GP1:90,2] + -0.066;
   1:L PR[91] R[100]mm/sec CNT100;
   1:  PR[GP1:91,1] = PR[GP1:90,1] + 48.439;
   1:  PR[GP1:91,2] = PR[GP1:90,2] + 7.543;
   1:L PR[91] R[100]mm/sec CNT100;
   1:  PR[GP1:91,1] = PR[GP1:90,1] + 47.383;
   1:  PR[GP1:91,2] = PR[GP1:90,2] + 14.212;
   1:L PR[91] R[100]mm/sec CNT100;
   1:  PR[GP1:91,1] = PR[GP1:90,1] + 44.280;
   1:  PR[GP1:91,2] = PR[GP1:90,2] + 21.239;
   1:L PR[91] R[100]mm/sec CNT100;
   1:  PR[GP1:91,1] = PR[GP1:90,1] + 41.215;
   1:  PR[GP1:91,2] = PR[GP1:90,2] + 27.256;
   1:L PR[91] R[100]mm/sec CNT100;
   1:  PR[GP1:91,1] = PR[GP1:90,1] + 36.308;
   1:  PR[GP1:91,2] = PR[GP1:90,2] + 33.166;
   1:L PR[91] R[100]mm/sec CNT100;
   1:  PR[GP1:91,1] = PR[GP1:90,1] + 31.530;
   1:  PR[GP1:91,2] = PR[GP1:90,2] + 37.944;
   1:L PR[91] R[100]mm/sec CNT100;
   1:  PR[GP1:91,1] = PR[GP1:90,1] + 25.959;
   1:  PR[GP1:91,2] = PR[GP1:90,2] + 41.889;
   1:L PR[91] R[100]mm/sec CNT100;
   1:  PR[GP1:91,1] = PR[GP1:90,1] + 19.934;
   1:  PR[GP1:91,2] = PR[GP1:90,2] + 44.959;
   1:L PR[91] R[100]mm/sec CNT100;
   1:  PR[GP1:91,1] = PR[GP1:90,1] + 13.569;
   1:  PR[GP1:91,2] = PR[GP1:90,2] + 47.425;
   1:L PR[91] R[100]mm/sec CNT100;
   1:  PR[GP1:91,1] = PR[GP1:90,1] + 6.890;
   1:  PR[GP1:91,2] = PR[GP1:90,2] + 48.483;
   1:L PR[91] R[100]mm/sec CNT100;
   1:  PR[GP1:91,1] = PR[GP1:90,1] + 0.105;
   1:  PR[GP1:91,2] = PR[GP1:90,2] + 49.323;
   1:L PR[91] R[100]mm/sec CNT100;
   1:  ! -- Layer/Ebene 218 -- !;
   1:  PR[91] = PR[90];
   1:  PR[GP1:91,1] = PR[GP1:90,1] + -5.934;
   1:  PR[GP1:91,2] = PR[GP1:90,2] + 48.575;
   1:  PR[GP1:91,3] = PR[GP1:90,3] + 133.285;
   1:L PR[91] R[100]mm/sec CNT100;
   1:  PR[GP1:91,1] = PR[GP1:90,1] + -13.556;
   1:  PR[GP1:91,2] = PR[GP1:90,2] + 47.368;
   1:L PR[91] R[100]mm/sec CNT100;
   1:  PR[GP1:91,1] = PR[GP1:90,1] + -19.220;
   1:  PR[GP1:91,2] = PR[GP1:90,2] + 45.173;
   1:L PR[91] R[100]mm/sec CNT100;
   1:  PR[GP1:91,1] = PR[GP1:90,1] + -26.095;
   1:  PR[GP1:91,2] = PR[GP1:90,2] + 41.670;
   1:L PR[91] R[100]mm/sec CNT100;
   1:  PR[GP1:91,1] = PR[GP1:90,1] + -31.053;
   1:  PR[GP1:91,2] = PR[GP1:90,2] + 38.159;
   1:L PR[91] R[100]mm/sec CNT100;
   1:  PR[GP1:91,1] = PR[GP1:90,1] + -36.507;
   1:  PR[GP1:91,2] = PR[GP1:90,2] + 32.705;
   1:L PR[91] R[100]mm/sec CNT100;
   1:  PR[GP1:91,1] = PR[GP1:90,1] + -40.875;
   1:  PR[GP1:91,2] = PR[GP1:90,2] + 27.444;
   1:L PR[91] R[100]mm/sec CNT100;
   1:  PR[GP1:91,1] = PR[GP1:90,1] + -44.374;
   1:  PR[GP1:91,2] = PR[GP1:90,2] + 20.577;
   1:L PR[91] R[100]mm/sec CNT100;
   1:  PR[GP1:91,1] = PR[GP1:90,1] + -47.134;
   1:  PR[GP1:91,2] = PR[GP1:90,2] + 14.325;
   1:L PR[91] R[100]mm/sec CNT100;
   1:  PR[GP1:91,1] = PR[GP1:90,1] + -48.081;
   1:  PR[GP1:91,2] = PR[GP1:90,2] + 7.534;
   1:L PR[91] R[100]mm/sec CNT100;
   1:  PR[GP1:91,1] = PR[GP1:90,1] + -49.287;
   1:  PR[GP1:91,2] = PR[GP1:90,2] + -0.078;
   1:L PR[91] R[100]mm/sec CNT100;
   1:  PR[GP1:91,1] = PR[GP1:90,1] + -48.342;
   1:  PR[GP1:91,2] = PR[GP1:90,2] + -6.852;
   1:L PR[91] R[100]mm/sec CNT100;
   1:  PR[GP1:91,1] = PR[GP1:90,1] + -47.136;
   1:  PR[GP1:91,2] = PR[GP1:90,2] + -14.464;
   1:L PR[91] R[100]mm/sec CNT100;
   1:  PR[GP1:91,1] = PR[GP1:90,1] + -44.374;
   1:  PR[GP1:91,2] = PR[GP1:90,2] + -20.721;
   1:L PR[91] R[100]mm/sec CNT100;
   1:  PR[GP1:91,1] = PR[GP1:90,1] + -40.875;
   1:  PR[GP1:91,2] = PR[GP1:90,2] + -27.588;
   1:L PR[91] R[100]mm/sec CNT100;
   1:  PR[GP1:91,1] = PR[GP1:90,1] + -36.507;
   1:  PR[GP1:91,2] = PR[GP1:90,2] + -32.849;
   1:L PR[91] R[100]mm/sec CNT100;
   1:  PR[GP1:91,1] = PR[GP1:90,1] + -31.053;
   1:  PR[GP1:91,2] = PR[GP1:90,2] + -38.303;
   1:L PR[91] R[100]mm/sec CNT100;
   1:  PR[GP1:91,1] = PR[GP1:90,1] + -26.095;
   1:  PR[GP1:91,2] = PR[GP1:90,2] + -41.814;
   1:L PR[91] R[100]mm/sec CNT100;
   1:  PR[GP1:91,1] = PR[GP1:90,1] + -19.220;
   1:  PR[GP1:91,2] = PR[GP1:90,2] + -45.317;
   1:L PR[91] R[100]mm/sec CNT100;
   1:  PR[GP1:91,1] = PR[GP1:90,1] + -13.565;
   1:  PR[GP1:91,2] = PR[GP1:90,2] + -47.508;
   1:L PR[91] R[100]mm/sec CNT100;
   1:  PR[GP1:91,1] = PR[GP1:90,1] + -7.505;
   1:  PR[GP1:91,2] = PR[GP1:90,2] + -48.259;
   1:L PR[91] R[100]mm/sec CNT100;
   1:  PR[GP1:91,1] = PR[GP1:90,1] + 0.116;
   1:  PR[GP1:91,2] = PR[GP1:90,2] + -49.466;
   1:L PR[91] R[100]mm/sec CNT100;
   1:  PR[GP1:91,1] = PR[GP1:90,1] + 6.146;
   1:  PR[GP1:91,2] = PR[GP1:90,2] + -48.719;
   1:L PR[91] R[100]mm/sec CNT100;
   1:  PR[GP1:91,1] = PR[GP1:90,1] + 13.768;
   1:  PR[GP1:91,2] = PR[GP1:90,2] + -47.512;
   1:L PR[91] R[100]mm/sec CNT100;
   1:  PR[GP1:91,1] = PR[GP1:90,1] + 19.433;
   1:  PR[GP1:91,2] = PR[GP1:90,2] + -45.317;
   1:L PR[91] R[100]mm/sec CNT100;
   1:  PR[GP1:91,1] = PR[GP1:90,1] + 26.309;
   1:  PR[GP1:91,2] = PR[GP1:90,2] + -41.814;
   1:L PR[91] R[100]mm/sec CNT100;
   1:  PR[GP1:91,1] = PR[GP1:90,1] + 31.268;
   1:  PR[GP1:91,2] = PR[GP1:90,2] + -38.302;
   1:L PR[91] R[100]mm/sec CNT100;
   1:  PR[GP1:91,1] = PR[GP1:90,1] + 36.720;
   1:  PR[GP1:91,2] = PR[GP1:90,2] + -32.849;
   1:L PR[91] R[100]mm/sec CNT100;
   1:  PR[GP1:91,1] = PR[GP1:90,1] + 41.089;
   1:  PR[GP1:91,2] = PR[GP1:90,2] + -27.587;
   1:L PR[91] R[100]mm/sec CNT100;
   1:  PR[GP1:91,1] = PR[GP1:90,1] + 44.587;
   1:  PR[GP1:91,2] = PR[GP1:90,2] + -20.720;
   1:L PR[91] R[100]mm/sec CNT100;
   1:  PR[GP1:91,1] = PR[GP1:90,1] + 47.347;
   1:  PR[GP1:91,2] = PR[GP1:90,2] + -14.469;
   1:L PR[91] R[100]mm/sec CNT100;
   1:  PR[GP1:91,1] = PR[GP1:90,1] + 48.294;
   1:  PR[GP1:91,2] = PR[GP1:90,2] + -7.678;
   1:L PR[91] R[100]mm/sec CNT100;
   1:  PR[GP1:91,1] = PR[GP1:90,1] + 49.500;
   1:  PR[GP1:91,2] = PR[GP1:90,2] + -0.066;
   1:L PR[91] R[100]mm/sec CNT100;
   1:  PR[GP1:91,1] = PR[GP1:90,1] + 48.555;
   1:  PR[GP1:91,2] = PR[GP1:90,2] + 6.708;
   1:L PR[91] R[100]mm/sec CNT100;
   1:  PR[GP1:91,1] = PR[GP1:90,1] + 47.350;
   1:  PR[GP1:91,2] = PR[GP1:90,2] + 14.320;
   1:L PR[91] R[100]mm/sec CNT100;
   1:  PR[GP1:91,1] = PR[GP1:90,1] + 44.588;
   1:  PR[GP1:91,2] = PR[GP1:90,2] + 20.576;
   1:L PR[91] R[100]mm/sec CNT100;
   1:  PR[GP1:91,1] = PR[GP1:90,1] + 41.089;
   1:  PR[GP1:91,2] = PR[GP1:90,2] + 27.443;
   1:L PR[91] R[100]mm/sec CNT100;
   1:  PR[GP1:91,1] = PR[GP1:90,1] + 36.720;
   1:  PR[GP1:91,2] = PR[GP1:90,2] + 32.706;
   1:L PR[91] R[100]mm/sec CNT100;
   1:  PR[GP1:91,1] = PR[GP1:90,1] + 31.268;
   1:  PR[GP1:91,2] = PR[GP1:90,2] + 38.158;
   1:L PR[91] R[100]mm/sec CNT100;
   1:  PR[GP1:91,1] = PR[GP1:90,1] + 26.309;
   1:  PR[GP1:91,2] = PR[GP1:90,2] + 41.670;
   1:L PR[91] R[100]mm/sec CNT100;
   1:  PR[GP1:91,1] = PR[GP1:90,1] + 19.433;
   1:  PR[GP1:91,2] = PR[GP1:90,2] + 45.173;
   1:L PR[91] R[100]mm/sec CNT100;
   1:  PR[GP1:91,1] = PR[GP1:90,1] + 13.768;
   1:  PR[GP1:91,2] = PR[GP1:90,2] + 47.368;
   1:L PR[91] R[100]mm/sec CNT100;
   1:  PR[GP1:91,1] = PR[GP1:90,1] + 6.146;
   1:  PR[GP1:91,2] = PR[GP1:90,2] + 48.575;
   1:L PR[91] R[100]mm/sec CNT100;
   1:  PR[GP1:91,1] = PR[GP1:90,1] + 0.106;
   1:  PR[GP1:91,2] = PR[GP1:90,2] + 49.323;
   1:L PR[91] R[100]mm/sec CNT100;
   1:  ! -- Layer/Ebene 219 -- !;
   1:  PR[91] = PR[90];
   1:  PR[GP1:91,1] = PR[GP1:90,1] + -5.190;
   1:  PR[GP1:91,2] = PR[GP1:90,2] + 48.667;
   1:  PR[GP1:91,3] = PR[GP1:90,3] + 133.895;
   1:L PR[91] R[100]mm/sec CNT100;
   1:  PR[GP1:91,1] = PR[GP1:90,1] + -13.754;
   1:  PR[GP1:91,2] = PR[GP1:90,2] + 47.311;
   1:L PR[91] R[100]mm/sec CNT100;
   1:  PR[GP1:91,1] = PR[GP1:90,1] + -18.719;
   1:  PR[GP1:91,2] = PR[GP1:90,2] + 45.387;
   1:L PR[91] R[100]mm/sec CNT100;
   1:  PR[GP1:91,1] = PR[GP1:90,1] + -26.445;
   1:  PR[GP1:91,2] = PR[GP1:90,2] + 41.450;
   1:L PR[91] R[100]mm/sec CNT100;
   1:  PR[GP1:91,1] = PR[GP1:90,1] + -30.791;
   1:  PR[GP1:91,2] = PR[GP1:90,2] + 38.373;
   1:L PR[91] R[100]mm/sec CNT100;
   1:  PR[GP1:91,1] = PR[GP1:90,1] + -36.919;
   1:  PR[GP1:91,2] = PR[GP1:90,2] + 32.244;
   1:L PR[91] R[100]mm/sec CNT100;
   1:  PR[GP1:91,1] = PR[GP1:90,1] + -40.749;
   1:  PR[GP1:91,2] = PR[GP1:90,2] + 27.631;
   1:L PR[91] R[100]mm/sec CNT100;
   1:  PR[GP1:91,1] = PR[GP1:90,1] + -44.681;
   1:  PR[GP1:91,2] = PR[GP1:90,2] + 19.914;
   1:L PR[91] R[100]mm/sec CNT100;
   1:  PR[GP1:91,1] = PR[GP1:90,1] + -47.101;
   1:  PR[GP1:91,2] = PR[GP1:90,2] + 14.433;
   1:L PR[91] R[100]mm/sec CNT100;
   1:  PR[GP1:91,1] = PR[GP1:90,1] + -47.932;
   1:  PR[GP1:91,2] = PR[GP1:90,2] + 8.476;
   1:L PR[91] R[100]mm/sec CNT100;
   1:  PR[GP1:91,1] = PR[GP1:90,1] + -49.287;
   1:  PR[GP1:91,2] = PR[GP1:90,2] + -0.078;
   1:L PR[91] R[100]mm/sec CNT100;
   1:  PR[GP1:91,1] = PR[GP1:90,1] + -48.458;
   1:  PR[GP1:91,2] = PR[GP1:90,2] + -6.018;
   1:L PR[91] R[100]mm/sec CNT100;
   1:  PR[GP1:91,1] = PR[GP1:90,1] + -47.103;
   1:  PR[GP1:91,2] = PR[GP1:90,2] + -14.572;
   1:L PR[91] R[100]mm/sec CNT100;
   1:  PR[GP1:91,1] = PR[GP1:90,1] + -44.681;
   1:  PR[GP1:91,2] = PR[GP1:90,2] + -20.058;
   1:L PR[91] R[100]mm/sec CNT100;
   1:  PR[GP1:91,1] = PR[GP1:90,1] + -40.749;
   1:  PR[GP1:91,2] = PR[GP1:90,2] + -27.775;
   1:L PR[91] R[100]mm/sec CNT100;
   1:  PR[GP1:91,1] = PR[GP1:90,1] + -36.919;
   1:  PR[GP1:91,2] = PR[GP1:90,2] + -32.388;
   1:L PR[91] R[100]mm/sec CNT100;
   1:  PR[GP1:91,1] = PR[GP1:90,1] + -30.791;
   1:  PR[GP1:91,2] = PR[GP1:90,2] + -38.517;
   1:L PR[91] R[100]mm/sec CNT100;
   1:  PR[GP1:91,1] = PR[GP1:90,1] + -26.445;
   1:  PR[GP1:91,2] = PR[GP1:90,2] + -41.594;
   1:L PR[91] R[100]mm/sec CNT100;
   1:  PR[GP1:91,1] = PR[GP1:90,1] + -18.719;
   1:  PR[GP1:91,2] = PR[GP1:90,2] + -45.531;
   1:L PR[91] R[100]mm/sec CNT100;
   1:  PR[GP1:91,1] = PR[GP1:90,1] + -13.763;
   1:  PR[GP1:91,2] = PR[GP1:90,2] + -47.451;
   1:L PR[91] R[100]mm/sec CNT100;
   1:  PR[GP1:91,1] = PR[GP1:90,1] + -8.448;
   1:  PR[GP1:91,2] = PR[GP1:90,2] + -48.110;
   1:L PR[91] R[100]mm/sec CNT100;
   1:  PR[GP1:91,1] = PR[GP1:90,1] + 0.116;
   1:  PR[GP1:91,2] = PR[GP1:90,2] + -49.466;
   1:L PR[91] R[100]mm/sec CNT100;
   1:  PR[GP1:91,1] = PR[GP1:90,1] + 5.402;
   1:  PR[GP1:91,2] = PR[GP1:90,2] + -48.811;
   1:L PR[91] R[100]mm/sec CNT100;
   1:  PR[GP1:91,1] = PR[GP1:90,1] + 13.966;
   1:  PR[GP1:91,2] = PR[GP1:90,2] + -47.455;
   1:L PR[91] R[100]mm/sec CNT100;
   1:  PR[GP1:91,1] = PR[GP1:90,1] + 18.932;
   1:  PR[GP1:91,2] = PR[GP1:90,2] + -45.531;
   1:L PR[91] R[100]mm/sec CNT100;
   1:  PR[GP1:91,1] = PR[GP1:90,1] + 26.658;
   1:  PR[GP1:91,2] = PR[GP1:90,2] + -41.594;
   1:L PR[91] R[100]mm/sec CNT100;
   1:  PR[GP1:91,1] = PR[GP1:90,1] + 31.005;
   1:  PR[GP1:91,2] = PR[GP1:90,2] + -38.516;
   1:L PR[91] R[100]mm/sec CNT100;
   1:  PR[GP1:91,1] = PR[GP1:90,1] + 37.133;
   1:  PR[GP1:91,2] = PR[GP1:90,2] + -32.389;
   1:L PR[91] R[100]mm/sec CNT100;
   1:  PR[GP1:91,1] = PR[GP1:90,1] + 40.963;
   1:  PR[GP1:91,2] = PR[GP1:90,2] + -27.774;
   1:L PR[91] R[100]mm/sec CNT100;
   1:  PR[GP1:91,1] = PR[GP1:90,1] + 44.895;
   1:  PR[GP1:91,2] = PR[GP1:90,2] + -20.058;
   1:L PR[91] R[100]mm/sec CNT100;
   1:  PR[GP1:91,1] = PR[GP1:90,1] + 47.314;
   1:  PR[GP1:91,2] = PR[GP1:90,2] + -14.577;
   1:L PR[91] R[100]mm/sec CNT100;
   1:  PR[GP1:91,1] = PR[GP1:90,1] + 48.145;
   1:  PR[GP1:91,2] = PR[GP1:90,2] + -8.620;
   1:L PR[91] R[100]mm/sec CNT100;
   1:  PR[GP1:91,1] = PR[GP1:90,1] + 49.500;
   1:  PR[GP1:91,2] = PR[GP1:90,2] + -0.066;
   1:L PR[91] R[100]mm/sec CNT100;
   1:  PR[GP1:91,1] = PR[GP1:90,1] + 48.672;
   1:  PR[GP1:91,2] = PR[GP1:90,2] + 5.873;
   1:L PR[91] R[100]mm/sec CNT100;
   1:  PR[GP1:91,1] = PR[GP1:90,1] + 47.317;
   1:  PR[GP1:91,2] = PR[GP1:90,2] + 14.427;
   1:L PR[91] R[100]mm/sec CNT100;
   1:  PR[GP1:91,1] = PR[GP1:90,1] + 44.895;
   1:  PR[GP1:91,2] = PR[GP1:90,2] + 19.913;
   1:L PR[91] R[100]mm/sec CNT100;
   1:  PR[GP1:91,1] = PR[GP1:90,1] + 40.963;
   1:  PR[GP1:91,2] = PR[GP1:90,2] + 27.631;
   1:L PR[91] R[100]mm/sec CNT100;
   1:  PR[GP1:91,1] = PR[GP1:90,1] + 37.133;
   1:  PR[GP1:91,2] = PR[GP1:90,2] + 32.245;
   1:L PR[91] R[100]mm/sec CNT100;
   1:  PR[GP1:91,1] = PR[GP1:90,1] + 31.005;
   1:  PR[GP1:91,2] = PR[GP1:90,2] + 38.372;
   1:L PR[91] R[100]mm/sec CNT100;
   1:  PR[GP1:91,1] = PR[GP1:90,1] + 26.658;
   1:  PR[GP1:91,2] = PR[GP1:90,2] + 41.450;
   1:L PR[91] R[100]mm/sec CNT100;
   1:  PR[GP1:91,1] = PR[GP1:90,1] + 18.932;
   1:  PR[GP1:91,2] = PR[GP1:90,2] + 45.387;
   1:L PR[91] R[100]mm/sec CNT100;
   1:  PR[GP1:91,1] = PR[GP1:90,1] + 13.966;
   1:  PR[GP1:91,2] = PR[GP1:90,2] + 47.311;
   1:L PR[91] R[100]mm/sec CNT100;
   1:  PR[GP1:91,1] = PR[GP1:90,1] + 5.402;
   1:  PR[GP1:91,2] = PR[GP1:90,2] + 48.667;
   1:L PR[91] R[100]mm/sec CNT100;
   1:  PR[GP1:91,1] = PR[GP1:90,1] + 0.106;
   1:  PR[GP1:91,2] = PR[GP1:90,2] + 49.323;
   1:L PR[91] R[100]mm/sec CNT100;
   1:  ! -- Layer/Ebene 220 -- !;
   1:  PR[91] = PR[90];
   1:  PR[GP1:91,1] = PR[GP1:90,1] + -4.446;
   1:  PR[GP1:91,2] = PR[GP1:90,2] + 48.759;
   1:  PR[GP1:91,3] = PR[GP1:90,3] + 134.505;
   1:L PR[91] R[100]mm/sec CNT100;
   1:  PR[GP1:91,1] = PR[GP1:90,1] + -13.952;
   1:  PR[GP1:91,2] = PR[GP1:90,2] + 47.254;
   1:L PR[91] R[100]mm/sec CNT100;
   1:  PR[GP1:91,1] = PR[GP1:90,1] + -18.219;
   1:  PR[GP1:91,2] = PR[GP1:90,2] + 45.600;
   1:L PR[91] R[100]mm/sec CNT100;
   1:  PR[GP1:91,1] = PR[GP1:90,1] + -26.794;
   1:  PR[GP1:91,2] = PR[GP1:90,2] + 41.231;
   1:L PR[91] R[100]mm/sec CNT100;
   1:  PR[GP1:91,1] = PR[GP1:90,1] + -30.529;
   1:  PR[GP1:91,2] = PR[GP1:90,2] + 38.587;
   1:L PR[91] R[100]mm/sec CNT100;
   1:  PR[GP1:91,1] = PR[GP1:90,1] + -37.332;
   1:  PR[GP1:91,2] = PR[GP1:90,2] + 31.783;
   1:L PR[91] R[100]mm/sec CNT100;
   1:  PR[GP1:91,1] = PR[GP1:90,1] + -40.624;
   1:  PR[GP1:91,2] = PR[GP1:90,2] + 27.818;
   1:L PR[91] R[100]mm/sec CNT100;
   1:  PR[GP1:91,1] = PR[GP1:90,1] + -44.989;
   1:  PR[GP1:91,2] = PR[GP1:90,2] + 19.251;
   1:L PR[91] R[100]mm/sec CNT100;
   1:  PR[GP1:91,1] = PR[GP1:90,1] + -47.068;
   1:  PR[GP1:91,2] = PR[GP1:90,2] + 14.541;
   1:L PR[91] R[100]mm/sec CNT100;
   1:  PR[GP1:91,1] = PR[GP1:90,1] + -47.783;
   1:  PR[GP1:91,2] = PR[GP1:90,2] + 9.419;
   1:L PR[91] R[100]mm/sec CNT100;
   1:  PR[GP1:91,1] = PR[GP1:90,1] + -49.287;
   1:  PR[GP1:91,2] = PR[GP1:90,2] + -0.078;
   1:L PR[91] R[100]mm/sec CNT100;
   1:  PR[GP1:91,1] = PR[GP1:90,1] + -48.575;
   1:  PR[GP1:91,2] = PR[GP1:90,2] + -5.183;
   1:L PR[91] R[100]mm/sec CNT100;
   1:  PR[GP1:91,1] = PR[GP1:90,1] + -47.071;
   1:  PR[GP1:91,2] = PR[GP1:90,2] + -14.680;
   1:L PR[91] R[100]mm/sec CNT100;
   1:  PR[GP1:91,1] = PR[GP1:90,1] + -44.989;
   1:  PR[GP1:91,2] = PR[GP1:90,2] + -19.395;
   1:L PR[91] R[100]mm/sec CNT100;
   1:  PR[GP1:91,1] = PR[GP1:90,1] + -40.624;
   1:  PR[GP1:91,2] = PR[GP1:90,2] + -27.962;
   1:L PR[91] R[100]mm/sec CNT100;
   1:  PR[GP1:91,1] = PR[GP1:90,1] + -37.332;
   1:  PR[GP1:91,2] = PR[GP1:90,2] + -31.927;
   1:L PR[91] R[100]mm/sec CNT100;
   1:  PR[GP1:91,1] = PR[GP1:90,1] + -30.529;
   1:  PR[GP1:91,2] = PR[GP1:90,2] + -38.731;
   1:L PR[91] R[100]mm/sec CNT100;
   1:  PR[GP1:91,1] = PR[GP1:90,1] + -26.794;
   1:  PR[GP1:91,2] = PR[GP1:90,2] + -41.375;
   1:L PR[91] R[100]mm/sec CNT100;
   1:  PR[GP1:91,1] = PR[GP1:90,1] + -18.219;
   1:  PR[GP1:91,2] = PR[GP1:90,2] + -45.744;
   1:L PR[91] R[100]mm/sec CNT100;
   1:  PR[GP1:91,1] = PR[GP1:90,1] + -13.962;
   1:  PR[GP1:91,2] = PR[GP1:90,2] + -47.394;
   1:L PR[91] R[100]mm/sec CNT100;
   1:  PR[GP1:91,1] = PR[GP1:90,1] + -9.390;
   1:  PR[GP1:91,2] = PR[GP1:90,2] + -47.961;
   1:L PR[91] R[100]mm/sec CNT100;
   1:  PR[GP1:91,1] = PR[GP1:90,1] + 0.116;
   1:  PR[GP1:91,2] = PR[GP1:90,2] + -49.466;
   1:L PR[91] R[100]mm/sec CNT100;
   1:  PR[GP1:91,1] = PR[GP1:90,1] + 4.658;
   1:  PR[GP1:91,2] = PR[GP1:90,2] + -48.904;
   1:L PR[91] R[100]mm/sec CNT100;
   1:  PR[GP1:91,1] = PR[GP1:90,1] + 14.165;
   1:  PR[GP1:91,2] = PR[GP1:90,2] + -47.398;
   1:L PR[91] R[100]mm/sec CNT100;
   1:  PR[GP1:91,1] = PR[GP1:90,1] + 18.432;
   1:  PR[GP1:91,2] = PR[GP1:90,2] + -45.744;
   1:L PR[91] R[100]mm/sec CNT100;
   1:  PR[GP1:91,1] = PR[GP1:90,1] + 27.008;
   1:  PR[GP1:91,2] = PR[GP1:90,2] + -41.375;
   1:L PR[91] R[100]mm/sec CNT100;
   1:  PR[GP1:91,1] = PR[GP1:90,1] + 30.743;
   1:  PR[GP1:91,2] = PR[GP1:90,2] + -38.730;
   1:L PR[91] R[100]mm/sec CNT100;
   1:  PR[GP1:91,1] = PR[GP1:90,1] + 37.545;
   1:  PR[GP1:91,2] = PR[GP1:90,2] + -31.928;
   1:L PR[91] R[100]mm/sec CNT100;
   1:  PR[GP1:91,1] = PR[GP1:90,1] + 40.837;
   1:  PR[GP1:91,2] = PR[GP1:90,2] + -27.962;
   1:L PR[91] R[100]mm/sec CNT100;
   1:  PR[GP1:91,1] = PR[GP1:90,1] + 45.202;
   1:  PR[GP1:91,2] = PR[GP1:90,2] + -19.395;
   1:L PR[91] R[100]mm/sec CNT100;
   1:  PR[GP1:91,1] = PR[GP1:90,1] + 47.282;
   1:  PR[GP1:91,2] = PR[GP1:90,2] + -14.685;
   1:L PR[91] R[100]mm/sec CNT100;
   1:  PR[GP1:91,1] = PR[GP1:90,1] + 47.996;
   1:  PR[GP1:91,2] = PR[GP1:90,2] + -9.563;
   1:L PR[91] R[100]mm/sec CNT100;
   1:  PR[GP1:91,1] = PR[GP1:90,1] + 49.500;
   1:  PR[GP1:91,2] = PR[GP1:90,2] + -0.066;
   1:L PR[91] R[100]mm/sec CNT100;
   1:  PR[GP1:91,1] = PR[GP1:90,1] + 48.788;
   1:  PR[GP1:91,2] = PR[GP1:90,2] + 5.039;
   1:L PR[91] R[100]mm/sec CNT100;
   1:  PR[GP1:91,1] = PR[GP1:90,1] + 47.284;
   1:  PR[GP1:91,2] = PR[GP1:90,2] + 14.535;
   1:L PR[91] R[100]mm/sec CNT100;
   1:  PR[GP1:91,1] = PR[GP1:90,1] + 45.202;
   1:  PR[GP1:91,2] = PR[GP1:90,2] + 19.251;
   1:L PR[91] R[100]mm/sec CNT100;
   1:  PR[GP1:91,1] = PR[GP1:90,1] + 40.837;
   1:  PR[GP1:91,2] = PR[GP1:90,2] + 27.818;
   1:L PR[91] R[100]mm/sec CNT100;
   1:  PR[GP1:91,1] = PR[GP1:90,1] + 37.545;
   1:  PR[GP1:91,2] = PR[GP1:90,2] + 31.784;
   1:L PR[91] R[100]mm/sec CNT100;
   1:  PR[GP1:91,1] = PR[GP1:90,1] + 30.743;
   1:  PR[GP1:91,2] = PR[GP1:90,2] + 38.586;
   1:L PR[91] R[100]mm/sec CNT100;
   1:  PR[GP1:91,1] = PR[GP1:90,1] + 27.008;
   1:  PR[GP1:91,2] = PR[GP1:90,2] + 41.231;
   1:L PR[91] R[100]mm/sec CNT100;
   1:  PR[GP1:91,1] = PR[GP1:90,1] + 18.432;
   1:  PR[GP1:91,2] = PR[GP1:90,2] + 45.600;
   1:L PR[91] R[100]mm/sec CNT100;
   1:  PR[GP1:91,1] = PR[GP1:90,1] + 14.165;
   1:  PR[GP1:91,2] = PR[GP1:90,2] + 47.254;
   1:L PR[91] R[100]mm/sec CNT100;
   1:  PR[GP1:91,1] = PR[GP1:90,1] + 4.658;
   1:  PR[GP1:91,2] = PR[GP1:90,2] + 48.760;
   1:L PR[91] R[100]mm/sec CNT100;
   1:  PR[GP1:91,1] = PR[GP1:90,1] + 0.106;
   1:  PR[GP1:91,2] = PR[GP1:90,2] + 49.323;
   1:L PR[91] R[100]mm/sec CNT100;
   1:  ! -- Layer/Ebene 221 -- !;
   1:  PR[91] = PR[90];
   1:  PR[GP1:91,1] = PR[GP1:90,1] + -3.702;
   1:  PR[GP1:91,2] = PR[GP1:90,2] + 48.852;
   1:  PR[GP1:91,3] = PR[GP1:90,3] + 135.115;
   1:L PR[91] R[100]mm/sec CNT100;
   1:  PR[GP1:91,1] = PR[GP1:90,1] + -14.150;
   1:  PR[GP1:91,2] = PR[GP1:90,2] + 47.197;
   1:L PR[91] R[100]mm/sec CNT100;
   1:  PR[GP1:91,1] = PR[GP1:90,1] + -17.718;
   1:  PR[GP1:91,2] = PR[GP1:90,2] + 45.814;
   1:L PR[91] R[100]mm/sec CNT100;
   1:  PR[GP1:91,1] = PR[GP1:90,1] + -27.144;
   1:  PR[GP1:91,2] = PR[GP1:90,2] + 41.011;
   1:L PR[91] R[100]mm/sec CNT100;
   1:  PR[GP1:91,1] = PR[GP1:90,1] + -30.266;
   1:  PR[GP1:91,2] = PR[GP1:90,2] + 38.800;
   1:L PR[91] R[100]mm/sec CNT100;
   1:  PR[GP1:91,1] = PR[GP1:90,1] + -37.744;
   1:  PR[GP1:91,2] = PR[GP1:90,2] + 31.323;
   1:L PR[91] R[100]mm/sec CNT100;
   1:  PR[GP1:91,1] = PR[GP1:90,1] + -40.498;
   1:  PR[GP1:91,2] = PR[GP1:90,2] + 28.006;
   1:L PR[91] R[100]mm/sec CNT100;
   1:  PR[GP1:91,1] = PR[GP1:90,1] + -45.296;
   1:  PR[GP1:91,2] = PR[GP1:90,2] + 18.588;
   1:L PR[91] R[100]mm/sec CNT100;
   1:  PR[GP1:91,1] = PR[GP1:90,1] + -47.035;
   1:  PR[GP1:91,2] = PR[GP1:90,2] + 14.649;
   1:L PR[91] R[100]mm/sec CNT100;
   1:  PR[GP1:91,1] = PR[GP1:90,1] + -47.633;
   1:  PR[GP1:91,2] = PR[GP1:90,2] + 10.362;
   1:L PR[91] R[100]mm/sec CNT100;
   1:  PR[GP1:91,1] = PR[GP1:90,1] + -49.287;
   1:  PR[GP1:91,2] = PR[GP1:90,2] + -0.078;
   1:L PR[91] R[100]mm/sec CNT100;
   1:  PR[GP1:91,1] = PR[GP1:90,1] + -48.691;
   1:  PR[GP1:91,2] = PR[GP1:90,2] + -4.348;
   1:L PR[91] R[100]mm/sec CNT100;
   1:  PR[GP1:91,1] = PR[GP1:90,1] + -47.038;
   1:  PR[GP1:91,2] = PR[GP1:90,2] + -14.787;
   1:L PR[91] R[100]mm/sec CNT100;
   1:  PR[GP1:91,1] = PR[GP1:90,1] + -45.296;
   1:  PR[GP1:91,2] = PR[GP1:90,2] + -18.732;
   1:L PR[91] R[100]mm/sec CNT100;
   1:  PR[GP1:91,1] = PR[GP1:90,1] + -40.498;
   1:  PR[GP1:91,2] = PR[GP1:90,2] + -28.150;
   1:L PR[91] R[100]mm/sec CNT100;
   1:  PR[GP1:91,1] = PR[GP1:90,1] + -37.744;
   1:  PR[GP1:91,2] = PR[GP1:90,2] + -31.467;
   1:L PR[91] R[100]mm/sec CNT100;
   1:  PR[GP1:91,1] = PR[GP1:90,1] + -30.266;
   1:  PR[GP1:91,2] = PR[GP1:90,2] + -38.944;
   1:L PR[91] R[100]mm/sec CNT100;
   1:  PR[GP1:91,1] = PR[GP1:90,1] + -27.144;
   1:  PR[GP1:91,2] = PR[GP1:90,2] + -41.155;
   1:L PR[91] R[100]mm/sec CNT100;
   1:  PR[GP1:91,1] = PR[GP1:90,1] + -17.718;
   1:  PR[GP1:91,2] = PR[GP1:90,2] + -45.958;
   1:L PR[91] R[100]mm/sec CNT100;
   1:  PR[GP1:91,1] = PR[GP1:90,1] + -14.160;
   1:  PR[GP1:91,2] = PR[GP1:90,2] + -47.337;
   1:L PR[91] R[100]mm/sec CNT100;
   1:  PR[GP1:91,1] = PR[GP1:90,1] + -10.332;
   1:  PR[GP1:91,2] = PR[GP1:90,2] + -47.811;
   1:L PR[91] R[100]mm/sec CNT100;
   1:  PR[GP1:91,1] = PR[GP1:90,1] + 0.116;
   1:  PR[GP1:91,2] = PR[GP1:90,2] + -49.466;
   1:L PR[91] R[100]mm/sec CNT100;
   1:  PR[GP1:91,1] = PR[GP1:90,1] + 3.914;
   1:  PR[GP1:91,2] = PR[GP1:90,2] + -48.996;
   1:L PR[91] R[100]mm/sec CNT100;
   1:  PR[GP1:91,1] = PR[GP1:90,1] + 14.363;
   1:  PR[GP1:91,2] = PR[GP1:90,2] + -47.341;
   1:L PR[91] R[100]mm/sec CNT100;
   1:  PR[GP1:91,1] = PR[GP1:90,1] + 17.931;
   1:  PR[GP1:91,2] = PR[GP1:90,2] + -45.958;
   1:L PR[91] R[100]mm/sec CNT100;
   1:  PR[GP1:91,1] = PR[GP1:90,1] + 27.357;
   1:  PR[GP1:91,2] = PR[GP1:90,2] + -41.155;
   1:L PR[91] R[100]mm/sec CNT100;
   1:  PR[GP1:91,1] = PR[GP1:90,1] + 30.480;
   1:  PR[GP1:91,2] = PR[GP1:90,2] + -38.944;
   1:L PR[91] R[100]mm/sec CNT100;
   1:  PR[GP1:91,1] = PR[GP1:90,1] + 37.957;
   1:  PR[GP1:91,2] = PR[GP1:90,2] + -31.467;
   1:L PR[91] R[100]mm/sec CNT100;
   1:  PR[GP1:91,1] = PR[GP1:90,1] + 40.711;
   1:  PR[GP1:91,2] = PR[GP1:90,2] + -28.149;
   1:L PR[91] R[100]mm/sec CNT100;
   1:  PR[GP1:91,1] = PR[GP1:90,1] + 45.510;
   1:  PR[GP1:91,2] = PR[GP1:90,2] + -18.732;
   1:L PR[91] R[100]mm/sec CNT100;
   1:  PR[GP1:91,1] = PR[GP1:90,1] + 47.249;
   1:  PR[GP1:91,2] = PR[GP1:90,2] + -14.793;
   1:L PR[91] R[100]mm/sec CNT100;
   1:  PR[GP1:91,1] = PR[GP1:90,1] + 47.847;
   1:  PR[GP1:91,2] = PR[GP1:90,2] + -10.505;
   1:L PR[91] R[100]mm/sec CNT100;
   1:  PR[GP1:91,1] = PR[GP1:90,1] + 49.500;
   1:  PR[GP1:91,2] = PR[GP1:90,2] + -0.066;
   1:L PR[91] R[100]mm/sec CNT100;
   1:  PR[GP1:91,1] = PR[GP1:90,1] + 48.904;
   1:  PR[GP1:91,2] = PR[GP1:90,2] + 4.204;
   1:L PR[91] R[100]mm/sec CNT100;
   1:  PR[GP1:91,1] = PR[GP1:90,1] + 47.251;
   1:  PR[GP1:91,2] = PR[GP1:90,2] + 14.643;
   1:L PR[91] R[100]mm/sec CNT100;
   1:  PR[GP1:91,1] = PR[GP1:90,1] + 45.510;
   1:  PR[GP1:91,2] = PR[GP1:90,2] + 18.588;
   1:L PR[91] R[100]mm/sec CNT100;
   1:  PR[GP1:91,1] = PR[GP1:90,1] + 40.711;
   1:  PR[GP1:91,2] = PR[GP1:90,2] + 28.005;
   1:L PR[91] R[100]mm/sec CNT100;
   1:  PR[GP1:91,1] = PR[GP1:90,1] + 37.957;
   1:  PR[GP1:91,2] = PR[GP1:90,2] + 31.323;
   1:L PR[91] R[100]mm/sec CNT100;
   1:  PR[GP1:91,1] = PR[GP1:90,1] + 30.480;
   1:  PR[GP1:91,2] = PR[GP1:90,2] + 38.800;
   1:L PR[91] R[100]mm/sec CNT100;
   1:  PR[GP1:91,1] = PR[GP1:90,1] + 27.357;
   1:  PR[GP1:91,2] = PR[GP1:90,2] + 41.011;
   1:L PR[91] R[100]mm/sec CNT100;
   1:  PR[GP1:91,1] = PR[GP1:90,1] + 17.931;
   1:  PR[GP1:91,2] = PR[GP1:90,2] + 45.814;
   1:L PR[91] R[100]mm/sec CNT100;
   1:  PR[GP1:91,1] = PR[GP1:90,1] + 14.363;
   1:  PR[GP1:91,2] = PR[GP1:90,2] + 47.197;
   1:L PR[91] R[100]mm/sec CNT100;
   1:  PR[GP1:91,1] = PR[GP1:90,1] + 3.914;
   1:  PR[GP1:91,2] = PR[GP1:90,2] + 48.852;
   1:L PR[91] R[100]mm/sec CNT100;
   1:  PR[GP1:91,1] = PR[GP1:90,1] + 0.106;
   1:  PR[GP1:91,2] = PR[GP1:90,2] + 49.323;
   1:L PR[91] R[100]mm/sec CNT100;
   1:  ! -- Layer/Ebene 222 -- !;
   1:  PR[91] = PR[90];
   1:  PR[GP1:91,1] = PR[GP1:90,1] + -2.958;
   1:  PR[GP1:91,2] = PR[GP1:90,2] + 48.944;
   1:  PR[GP1:91,3] = PR[GP1:90,3] + 135.725;
   1:L PR[91] R[100]mm/sec CNT100;
   1:  PR[GP1:91,1] = PR[GP1:90,1] + -14.349;
   1:  PR[GP1:91,2] = PR[GP1:90,2] + 47.140;
   1:L PR[91] R[100]mm/sec CNT100;
   1:  PR[GP1:91,1] = PR[GP1:90,1] + -17.217;
   1:  PR[GP1:91,2] = PR[GP1:90,2] + 46.028;
   1:L PR[91] R[100]mm/sec CNT100;
   1:  PR[GP1:91,1] = PR[GP1:90,1] + -27.493;
   1:  PR[GP1:91,2] = PR[GP1:90,2] + 40.792;
   1:L PR[91] R[100]mm/sec CNT100;
   1:  PR[GP1:91,1] = PR[GP1:90,1] + -30.004;
   1:  PR[GP1:91,2] = PR[GP1:90,2] + 39.014;
   1:L PR[91] R[100]mm/sec CNT100;
   1:  PR[GP1:91,1] = PR[GP1:90,1] + -38.156;
   1:  PR[GP1:91,2] = PR[GP1:90,2] + 30.862;
   1:L PR[91] R[100]mm/sec CNT100;
   1:  PR[GP1:91,1] = PR[GP1:90,1] + -40.372;
   1:  PR[GP1:91,2] = PR[GP1:90,2] + 28.193;
   1:L PR[91] R[100]mm/sec CNT100;
   1:  PR[GP1:91,1] = PR[GP1:90,1] + -45.604;
   1:  PR[GP1:91,2] = PR[GP1:90,2] + 17.925;
   1:L PR[91] R[100]mm/sec CNT100;
   1:  PR[GP1:91,1] = PR[GP1:90,1] + -47.003;
   1:  PR[GP1:91,2] = PR[GP1:90,2] + 14.757;
   1:L PR[91] R[100]mm/sec CNT100;
   1:  PR[GP1:91,1] = PR[GP1:90,1] + -47.484;
   1:  PR[GP1:91,2] = PR[GP1:90,2] + 11.304;
   1:L PR[91] R[100]mm/sec CNT100;
   1:  PR[GP1:91,1] = PR[GP1:90,1] + -49.287;
   1:  PR[GP1:91,2] = PR[GP1:90,2] + -0.078;
   1:L PR[91] R[100]mm/sec CNT100;
   1:  PR[GP1:91,1] = PR[GP1:90,1] + -48.807;
   1:  PR[GP1:91,2] = PR[GP1:90,2] + -3.514;
   1:L PR[91] R[100]mm/sec CNT100;
   1:  PR[GP1:91,1] = PR[GP1:90,1] + -47.005;
   1:  PR[GP1:91,2] = PR[GP1:90,2] + -14.895;
   1:L PR[91] R[100]mm/sec CNT100;
   1:  PR[GP1:91,1] = PR[GP1:90,1] + -45.604;
   1:  PR[GP1:91,2] = PR[GP1:90,2] + -18.069;
   1:L PR[91] R[100]mm/sec CNT100;
   1:  PR[GP1:91,1] = PR[GP1:90,1] + -40.372;
   1:  PR[GP1:91,2] = PR[GP1:90,2] + -28.337;
   1:L PR[91] R[100]mm/sec CNT100;
   1:  PR[GP1:91,1] = PR[GP1:90,1] + -38.156;
   1:  PR[GP1:91,2] = PR[GP1:90,2] + -31.006;
   1:L PR[91] R[100]mm/sec CNT100;
   1:  PR[GP1:91,1] = PR[GP1:90,1] + -30.004;
   1:  PR[GP1:91,2] = PR[GP1:90,2] + -39.158;
   1:L PR[91] R[100]mm/sec CNT100;
   1:  PR[GP1:91,1] = PR[GP1:90,1] + -27.493;
   1:  PR[GP1:91,2] = PR[GP1:90,2] + -40.936;
   1:L PR[91] R[100]mm/sec CNT100;
   1:  PR[GP1:91,1] = PR[GP1:90,1] + -17.217;
   1:  PR[GP1:91,2] = PR[GP1:90,2] + -46.172;
   1:L PR[91] R[100]mm/sec CNT100;
   1:  PR[GP1:91,1] = PR[GP1:90,1] + -14.358;
   1:  PR[GP1:91,2] = PR[GP1:90,2] + -47.280;
   1:L PR[91] R[100]mm/sec CNT100;
   1:  PR[GP1:91,1] = PR[GP1:90,1] + -11.275;
   1:  PR[GP1:91,2] = PR[GP1:90,2] + -47.662;
   1:L PR[91] R[100]mm/sec CNT100;
   1:  PR[GP1:91,1] = PR[GP1:90,1] + 0.116;
   1:  PR[GP1:91,2] = PR[GP1:90,2] + -49.466;
   1:L PR[91] R[100]mm/sec CNT100;
   1:  PR[GP1:91,1] = PR[GP1:90,1] + 3.170;
   1:  PR[GP1:91,2] = PR[GP1:90,2] + -49.088;
   1:L PR[91] R[100]mm/sec CNT100;
   1:  PR[GP1:91,1] = PR[GP1:90,1] + 14.561;
   1:  PR[GP1:91,2] = PR[GP1:90,2] + -47.284;
   1:L PR[91] R[100]mm/sec CNT100;
   1:  PR[GP1:91,1] = PR[GP1:90,1] + 17.430;
   1:  PR[GP1:91,2] = PR[GP1:90,2] + -46.172;
   1:L PR[91] R[100]mm/sec CNT100;
   1:  PR[GP1:91,1] = PR[GP1:90,1] + 27.707;
   1:  PR[GP1:91,2] = PR[GP1:90,2] + -40.936;
   1:L PR[91] R[100]mm/sec CNT100;
   1:  PR[GP1:91,1] = PR[GP1:90,1] + 30.218;
   1:  PR[GP1:91,2] = PR[GP1:90,2] + -39.158;
   1:L PR[91] R[100]mm/sec CNT100;
   1:  PR[GP1:91,1] = PR[GP1:90,1] + 38.370;
   1:  PR[GP1:91,2] = PR[GP1:90,2] + -31.006;
   1:L PR[91] R[100]mm/sec CNT100;
   1:  PR[GP1:91,1] = PR[GP1:90,1] + 40.585;
   1:  PR[GP1:91,2] = PR[GP1:90,2] + -28.337;
   1:L PR[91] R[100]mm/sec CNT100;
   1:  PR[GP1:91,1] = PR[GP1:90,1] + 45.817;
   1:  PR[GP1:91,2] = PR[GP1:90,2] + -18.069;
   1:L PR[91] R[100]mm/sec CNT100;
   1:  PR[GP1:91,1] = PR[GP1:90,1] + 47.216;
   1:  PR[GP1:91,2] = PR[GP1:90,2] + -14.900;
   1:L PR[91] R[100]mm/sec CNT100;
   1:  PR[GP1:91,1] = PR[GP1:90,1] + 47.697;
   1:  PR[GP1:91,2] = PR[GP1:90,2] + -11.448;
   1:L PR[91] R[100]mm/sec CNT100;
   1:  PR[GP1:91,1] = PR[GP1:90,1] + 49.500;
   1:  PR[GP1:91,2] = PR[GP1:90,2] + -0.066;
   1:L PR[91] R[100]mm/sec CNT100;
   1:  PR[GP1:91,1] = PR[GP1:90,1] + 49.021;
   1:  PR[GP1:91,2] = PR[GP1:90,2] + 3.370;
   1:L PR[91] R[100]mm/sec CNT100;
   1:  PR[GP1:91,1] = PR[GP1:90,1] + 47.218;
   1:  PR[GP1:91,2] = PR[GP1:90,2] + 14.751;
   1:L PR[91] R[100]mm/sec CNT100;
   1:  PR[GP1:91,1] = PR[GP1:90,1] + 45.817;
   1:  PR[GP1:91,2] = PR[GP1:90,2] + 17.925;
   1:L PR[91] R[100]mm/sec CNT100;
   1:  PR[GP1:91,1] = PR[GP1:90,1] + 40.585;
   1:  PR[GP1:91,2] = PR[GP1:90,2] + 28.193;
   1:L PR[91] R[100]mm/sec CNT100;
   1:  PR[GP1:91,1] = PR[GP1:90,1] + 38.370;
   1:  PR[GP1:91,2] = PR[GP1:90,2] + 30.862;
   1:L PR[91] R[100]mm/sec CNT100;
   1:  PR[GP1:91,1] = PR[GP1:90,1] + 30.218;
   1:  PR[GP1:91,2] = PR[GP1:90,2] + 39.014;
   1:L PR[91] R[100]mm/sec CNT100;
   1:  PR[GP1:91,1] = PR[GP1:90,1] + 27.706;
   1:  PR[GP1:91,2] = PR[GP1:90,2] + 40.792;
   1:L PR[91] R[100]mm/sec CNT100;
   1:  PR[GP1:91,1] = PR[GP1:90,1] + 17.430;
   1:  PR[GP1:91,2] = PR[GP1:90,2] + 46.028;
   1:L PR[91] R[100]mm/sec CNT100;
   1:  PR[GP1:91,1] = PR[GP1:90,1] + 14.561;
   1:  PR[GP1:91,2] = PR[GP1:90,2] + 47.140;
   1:L PR[91] R[100]mm/sec CNT100;
   1:  PR[GP1:91,1] = PR[GP1:90,1] + 3.170;
   1:  PR[GP1:91,2] = PR[GP1:90,2] + 48.944;
   1:L PR[91] R[100]mm/sec CNT100;
   1:  PR[GP1:91,1] = PR[GP1:90,1] + 0.106;
   1:  PR[GP1:91,2] = PR[GP1:90,2] + 49.323;
   1:L PR[91] R[100]mm/sec CNT100;
   1:  ! -- Layer/Ebene 223 -- !;
   1:  PR[91] = PR[90];
   1:  PR[GP1:91,1] = PR[GP1:90,1] + -2.213;
   1:  PR[GP1:91,2] = PR[GP1:90,2] + 49.036;
   1:  PR[GP1:91,3] = PR[GP1:90,3] + 136.335;
   1:L PR[91] R[100]mm/sec CNT100;
   1:  PR[GP1:91,1] = PR[GP1:90,1] + -14.547;
   1:  PR[GP1:91,2] = PR[GP1:90,2] + 47.083;
   1:L PR[91] R[100]mm/sec CNT100;
   1:  PR[GP1:91,1] = PR[GP1:90,1] + -16.716;
   1:  PR[GP1:91,2] = PR[GP1:90,2] + 46.242;
   1:L PR[91] R[100]mm/sec CNT100;
   1:  PR[GP1:91,1] = PR[GP1:90,1] + -27.843;
   1:  PR[GP1:91,2] = PR[GP1:90,2] + 40.573;
   1:L PR[91] R[100]mm/sec CNT100;
   1:  PR[GP1:91,1] = PR[GP1:90,1] + -29.742;
   1:  PR[GP1:91,2] = PR[GP1:90,2] + 39.228;
   1:L PR[91] R[100]mm/sec CNT100;
   1:  PR[GP1:91,1] = PR[GP1:90,1] + -38.569;
   1:  PR[GP1:91,2] = PR[GP1:90,2] + 30.401;
   1:L PR[91] R[100]mm/sec CNT100;
   1:  PR[GP1:91,1] = PR[GP1:90,1] + -40.246;
   1:  PR[GP1:91,2] = PR[GP1:90,2] + 28.380;
   1:L PR[91] R[100]mm/sec CNT100;
   1:  PR[GP1:91,1] = PR[GP1:90,1] + -45.911;
   1:  PR[GP1:91,2] = PR[GP1:90,2] + 17.262;
   1:L PR[91] R[100]mm/sec CNT100;
   1:  PR[GP1:91,1] = PR[GP1:90,1] + -46.970;
   1:  PR[GP1:91,2] = PR[GP1:90,2] + 14.865;
   1:L PR[91] R[100]mm/sec CNT100;
   1:  PR[GP1:91,1] = PR[GP1:90,1] + -47.335;
   1:  PR[GP1:91,2] = PR[GP1:90,2] + 12.247;
   1:L PR[91] R[100]mm/sec CNT100;
   1:  PR[GP1:91,1] = PR[GP1:90,1] + -49.287;
   1:  PR[GP1:91,2] = PR[GP1:90,2] + -0.078;
   1:L PR[91] R[100]mm/sec CNT100;
   1:  PR[GP1:91,1] = PR[GP1:90,1] + -48.924;
   1:  PR[GP1:91,2] = PR[GP1:90,2] + -2.679;
   1:L PR[91] R[100]mm/sec CNT100;
   1:  PR[GP1:91,1] = PR[GP1:90,1] + -46.972;
   1:  PR[GP1:91,2] = PR[GP1:90,2] + -15.003;
   1:L PR[91] R[100]mm/sec CNT100;
   1:  PR[GP1:91,1] = PR[GP1:90,1] + -45.911;
   1:  PR[GP1:91,2] = PR[GP1:90,2] + -17.406;
   1:L PR[91] R[100]mm/sec CNT100;
   1:  PR[GP1:91,1] = PR[GP1:90,1] + -40.246;
   1:  PR[GP1:91,2] = PR[GP1:90,2] + -28.524;
   1:L PR[91] R[100]mm/sec CNT100;
   1:  PR[GP1:91,1] = PR[GP1:90,1] + -38.569;
   1:  PR[GP1:91,2] = PR[GP1:90,2] + -30.545;
   1:L PR[91] R[100]mm/sec CNT100;
   1:  PR[GP1:91,1] = PR[GP1:90,1] + -29.742;
   1:  PR[GP1:91,2] = PR[GP1:90,2] + -39.372;
   1:L PR[91] R[100]mm/sec CNT100;
   1:  PR[GP1:91,1] = PR[GP1:90,1] + -27.843;
   1:  PR[GP1:91,2] = PR[GP1:90,2] + -40.717;
   1:L PR[91] R[100]mm/sec CNT100;
   1:  PR[GP1:91,1] = PR[GP1:90,1] + -16.716;
   1:  PR[GP1:91,2] = PR[GP1:90,2] + -46.386;
   1:L PR[91] R[100]mm/sec CNT100;
   1:  PR[GP1:91,1] = PR[GP1:90,1] + -14.556;
   1:  PR[GP1:91,2] = PR[GP1:90,2] + -47.223;
   1:L PR[91] R[100]mm/sec CNT100;
   1:  PR[GP1:91,1] = PR[GP1:90,1] + -12.217;
   1:  PR[GP1:91,2] = PR[GP1:90,2] + -47.513;
   1:L PR[91] R[100]mm/sec CNT100;
   1:  PR[GP1:91,1] = PR[GP1:90,1] + 0.116;
   1:  PR[GP1:91,2] = PR[GP1:90,2] + -49.466;
   1:L PR[91] R[100]mm/sec CNT100;
   1:  PR[GP1:91,1] = PR[GP1:90,1] + 2.426;
   1:  PR[GP1:91,2] = PR[GP1:90,2] + -49.180;
   1:L PR[91] R[100]mm/sec CNT100;
   1:  PR[GP1:91,1] = PR[GP1:90,1] + 14.760;
   1:  PR[GP1:91,2] = PR[GP1:90,2] + -47.227;
   1:L PR[91] R[100]mm/sec CNT100;
   1:  PR[GP1:91,1] = PR[GP1:90,1] + 16.930;
   1:  PR[GP1:91,2] = PR[GP1:90,2] + -46.386;
   1:L PR[91] R[100]mm/sec CNT100;
   1:  PR[GP1:91,1] = PR[GP1:90,1] + 28.056;
   1:  PR[GP1:91,2] = PR[GP1:90,2] + -40.717;
   1:L PR[91] R[100]mm/sec CNT100;
   1:  PR[GP1:91,1] = PR[GP1:90,1] + 29.955;
   1:  PR[GP1:91,2] = PR[GP1:90,2] + -39.372;
   1:L PR[91] R[100]mm/sec CNT100;
   1:  PR[GP1:91,1] = PR[GP1:90,1] + 38.782;
   1:  PR[GP1:91,2] = PR[GP1:90,2] + -30.545;
   1:L PR[91] R[100]mm/sec CNT100;
   1:  PR[GP1:91,1] = PR[GP1:90,1] + 40.460;
   1:  PR[GP1:91,2] = PR[GP1:90,2] + -28.524;
   1:L PR[91] R[100]mm/sec CNT100;
   1:  PR[GP1:91,1] = PR[GP1:90,1] + 46.124;
   1:  PR[GP1:91,2] = PR[GP1:90,2] + -17.406;
   1:L PR[91] R[100]mm/sec CNT100;
   1:  PR[GP1:91,1] = PR[GP1:90,1] + 47.183;
   1:  PR[GP1:91,2] = PR[GP1:90,2] + -15.008;
   1:L PR[91] R[100]mm/sec CNT100;
   1:  PR[GP1:91,1] = PR[GP1:90,1] + 47.548;
   1:  PR[GP1:91,2] = PR[GP1:90,2] + -12.390;
   1:L PR[91] R[100]mm/sec CNT100;
   1:  PR[GP1:91,1] = PR[GP1:90,1] + 49.500;
   1:  PR[GP1:91,2] = PR[GP1:90,2] + -0.066;
   1:L PR[91] R[100]mm/sec CNT100;
   1:  PR[GP1:91,1] = PR[GP1:90,1] + 49.137;
   1:  PR[GP1:91,2] = PR[GP1:90,2] + 2.535;
   1:L PR[91] R[100]mm/sec CNT100;
   1:  PR[GP1:91,1] = PR[GP1:90,1] + 47.185;
   1:  PR[GP1:91,2] = PR[GP1:90,2] + 14.859;
   1:L PR[91] R[100]mm/sec CNT100;
   1:  PR[GP1:91,1] = PR[GP1:90,1] + 46.125;
   1:  PR[GP1:91,2] = PR[GP1:90,2] + 17.262;
   1:L PR[91] R[100]mm/sec CNT100;
   1:  PR[GP1:91,1] = PR[GP1:90,1] + 40.460;
   1:  PR[GP1:91,2] = PR[GP1:90,2] + 28.380;
   1:L PR[91] R[100]mm/sec CNT100;
   1:  PR[GP1:91,1] = PR[GP1:90,1] + 38.782;
   1:  PR[GP1:91,2] = PR[GP1:90,2] + 30.401;
   1:L PR[91] R[100]mm/sec CNT100;
   1:  PR[GP1:91,1] = PR[GP1:90,1] + 29.955;
   1:  PR[GP1:91,2] = PR[GP1:90,2] + 39.228;
   1:L PR[91] R[100]mm/sec CNT100;
   1:  PR[GP1:91,1] = PR[GP1:90,1] + 28.056;
   1:  PR[GP1:91,2] = PR[GP1:90,2] + 40.573;
   1:L PR[91] R[100]mm/sec CNT100;
   1:  PR[GP1:91,1] = PR[GP1:90,1] + 16.929;
   1:  PR[GP1:91,2] = PR[GP1:90,2] + 46.242;
   1:L PR[91] R[100]mm/sec CNT100;
   1:  PR[GP1:91,1] = PR[GP1:90,1] + 14.760;
   1:  PR[GP1:91,2] = PR[GP1:90,2] + 47.083;
   1:L PR[91] R[100]mm/sec CNT100;
   1:  PR[GP1:91,1] = PR[GP1:90,1] + 2.426;
   1:  PR[GP1:91,2] = PR[GP1:90,2] + 49.036;
   1:L PR[91] R[100]mm/sec CNT100;
   1:  PR[GP1:91,1] = PR[GP1:90,1] + 0.106;
   1:  PR[GP1:91,2] = PR[GP1:90,2] + 49.323;
   1:L PR[91] R[100]mm/sec CNT100;
   1:  ! -- Layer/Ebene 224 -- !;
   1:  PR[91] = PR[90];
   1:  PR[GP1:91,1] = PR[GP1:90,1] + -1.469;
   1:  PR[GP1:91,2] = PR[GP1:90,2] + 49.128;
   1:  PR[GP1:91,3] = PR[GP1:90,3] + 136.945;
   1:L PR[91] R[100]mm/sec CNT100;
   1:  PR[GP1:91,1] = PR[GP1:90,1] + -14.745;
   1:  PR[GP1:91,2] = PR[GP1:90,2] + 47.025;
   1:L PR[91] R[100]mm/sec CNT100;
   1:  PR[GP1:91,1] = PR[GP1:90,1] + -16.215;
   1:  PR[GP1:91,2] = PR[GP1:90,2] + 46.456;
   1:L PR[91] R[100]mm/sec CNT100;
   1:  PR[GP1:91,1] = PR[GP1:90,1] + -28.192;
   1:  PR[GP1:91,2] = PR[GP1:90,2] + 40.353;
   1:L PR[91] R[100]mm/sec CNT100;
   1:  PR[GP1:91,1] = PR[GP1:90,1] + -29.479;
   1:  PR[GP1:91,2] = PR[GP1:90,2] + 39.442;
   1:L PR[91] R[100]mm/sec CNT100;
   1:  PR[GP1:91,1] = PR[GP1:90,1] + -38.981;
   1:  PR[GP1:91,2] = PR[GP1:90,2] + 29.940;
   1:L PR[91] R[100]mm/sec CNT100;
   1:  PR[GP1:91,1] = PR[GP1:90,1] + -40.120;
   1:  PR[GP1:91,2] = PR[GP1:90,2] + 28.568;
   1:L PR[91] R[100]mm/sec CNT100;
   1:  PR[GP1:91,1] = PR[GP1:90,1] + -46.219;
   1:  PR[GP1:91,2] = PR[GP1:90,2] + 16.599;
   1:L PR[91] R[100]mm/sec CNT100;
   1:  PR[GP1:91,1] = PR[GP1:90,1] + -46.937;
   1:  PR[GP1:91,2] = PR[GP1:90,2] + 14.972;
   1:L PR[91] R[100]mm/sec CNT100;
   1:  PR[GP1:91,1] = PR[GP1:90,1] + -47.185;
   1:  PR[GP1:91,2] = PR[GP1:90,2] + 13.189;
   1:L PR[91] R[100]mm/sec CNT100;
   1:  PR[GP1:91,1] = PR[GP1:90,1] + -49.287;
   1:  PR[GP1:91,2] = PR[GP1:90,2] + -0.078;
   1:L PR[91] R[100]mm/sec CNT100;
   1:  PR[GP1:91,1] = PR[GP1:90,1] + -49.040;
   1:  PR[GP1:91,2] = PR[GP1:90,2] + -1.845;
   1:L PR[91] R[100]mm/sec CNT100;
   1:  PR[GP1:91,1] = PR[GP1:90,1] + -46.939;
   1:  PR[GP1:91,2] = PR[GP1:90,2] + -15.111;
   1:L PR[91] R[100]mm/sec CNT100;
   1:  PR[GP1:91,1] = PR[GP1:90,1] + -46.219;
   1:  PR[GP1:91,2] = PR[GP1:90,2] + -16.743;
   1:L PR[91] R[100]mm/sec CNT100;
   1:  PR[GP1:91,1] = PR[GP1:90,1] + -40.120;
   1:  PR[GP1:91,2] = PR[GP1:90,2] + -28.712;
   1:L PR[91] R[100]mm/sec CNT100;
   1:  PR[GP1:91,1] = PR[GP1:90,1] + -38.981;
   1:  PR[GP1:91,2] = PR[GP1:90,2] + -30.084;
   1:L PR[91] R[100]mm/sec CNT100;
   1:  PR[GP1:91,1] = PR[GP1:90,1] + -29.479;
   1:  PR[GP1:91,2] = PR[GP1:90,2] + -39.586;
   1:L PR[91] R[100]mm/sec CNT100;
   1:  PR[GP1:91,1] = PR[GP1:90,1] + -28.192;
   1:  PR[GP1:91,2] = PR[GP1:90,2] + -40.497;
   1:L PR[91] R[100]mm/sec CNT100;
   1:  PR[GP1:91,1] = PR[GP1:90,1] + -16.216;
   1:  PR[GP1:91,2] = PR[GP1:90,2] + -46.600;
   1:L PR[91] R[100]mm/sec CNT100;
   1:  PR[GP1:91,1] = PR[GP1:90,1] + -14.755;
   1:  PR[GP1:91,2] = PR[GP1:90,2] + -47.166;
   1:L PR[91] R[100]mm/sec CNT100;
   1:  PR[GP1:91,1] = PR[GP1:90,1] + -13.159;
   1:  PR[GP1:91,2] = PR[GP1:90,2] + -47.363;
   1:L PR[91] R[100]mm/sec CNT100;
   1:  PR[GP1:91,1] = PR[GP1:90,1] + 0.117;
   1:  PR[GP1:91,2] = PR[GP1:90,2] + -49.466;
   1:L PR[91] R[100]mm/sec CNT100;
   1:  PR[GP1:91,1] = PR[GP1:90,1] + 1.682;
   1:  PR[GP1:91,2] = PR[GP1:90,2] + -49.272;
   1:L PR[91] R[100]mm/sec CNT100;
   1:  PR[GP1:91,1] = PR[GP1:90,1] + 14.958;
   1:  PR[GP1:91,2] = PR[GP1:90,2] + -47.170;
   1:L PR[91] R[100]mm/sec CNT100;
   1:  PR[GP1:91,1] = PR[GP1:90,1] + 16.429;
   1:  PR[GP1:91,2] = PR[GP1:90,2] + -46.600;
   1:L PR[91] R[100]mm/sec CNT100;
   1:  PR[GP1:91,1] = PR[GP1:90,1] + 28.405;
   1:  PR[GP1:91,2] = PR[GP1:90,2] + -40.497;
   1:L PR[91] R[100]mm/sec CNT100;
   1:  PR[GP1:91,1] = PR[GP1:90,1] + 29.693;
   1:  PR[GP1:91,2] = PR[GP1:90,2] + -39.586;
   1:L PR[91] R[100]mm/sec CNT100;
   1:  PR[GP1:91,1] = PR[GP1:90,1] + 39.194;
   1:  PR[GP1:91,2] = PR[GP1:90,2] + -30.084;
   1:L PR[91] R[100]mm/sec CNT100;
   1:  PR[GP1:91,1] = PR[GP1:90,1] + 40.334;
   1:  PR[GP1:91,2] = PR[GP1:90,2] + -28.712;
   1:L PR[91] R[100]mm/sec CNT100;
   1:  PR[GP1:91,1] = PR[GP1:90,1] + 46.432;
   1:  PR[GP1:91,2] = PR[GP1:90,2] + -16.743;
   1:L PR[91] R[100]mm/sec CNT100;
   1:  PR[GP1:91,1] = PR[GP1:90,1] + 47.150;
   1:  PR[GP1:91,2] = PR[GP1:90,2] + -15.116;
   1:L PR[91] R[100]mm/sec CNT100;
   1:  PR[GP1:91,1] = PR[GP1:90,1] + 47.399;
   1:  PR[GP1:91,2] = PR[GP1:90,2] + -13.333;
   1:L PR[91] R[100]mm/sec CNT100;
   1:  PR[GP1:91,1] = PR[GP1:90,1] + 49.500;
   1:  PR[GP1:91,2] = PR[GP1:90,2] + -0.066;
   1:L PR[91] R[100]mm/sec CNT100;
   1:  PR[GP1:91,1] = PR[GP1:90,1] + 49.254;
   1:  PR[GP1:91,2] = PR[GP1:90,2] + 1.701;
   1:L PR[91] R[100]mm/sec CNT100;
   1:  PR[GP1:91,1] = PR[GP1:90,1] + 47.152;
   1:  PR[GP1:91,2] = PR[GP1:90,2] + 14.967;
   1:L PR[91] R[100]mm/sec CNT100;
   1:  PR[GP1:91,1] = PR[GP1:90,1] + 46.432;
   1:  PR[GP1:91,2] = PR[GP1:90,2] + 16.599;
   1:L PR[91] R[100]mm/sec CNT100;
   1:  PR[GP1:91,1] = PR[GP1:90,1] + 40.334;
   1:  PR[GP1:91,2] = PR[GP1:90,2] + 28.568;
   1:L PR[91] R[100]mm/sec CNT100;
   1:  PR[GP1:91,1] = PR[GP1:90,1] + 39.194;
   1:  PR[GP1:91,2] = PR[GP1:90,2] + 29.940;
   1:L PR[91] R[100]mm/sec CNT100;
   1:  PR[GP1:91,1] = PR[GP1:90,1] + 29.693;
   1:  PR[GP1:91,2] = PR[GP1:90,2] + 39.442;
   1:L PR[91] R[100]mm/sec CNT100;
   1:  PR[GP1:91,1] = PR[GP1:90,1] + 28.405;
   1:  PR[GP1:91,2] = PR[GP1:90,2] + 40.353;
   1:L PR[91] R[100]mm/sec CNT100;
   1:  PR[GP1:91,1] = PR[GP1:90,1] + 16.429;
   1:  PR[GP1:91,2] = PR[GP1:90,2] + 46.456;
   1:L PR[91] R[100]mm/sec CNT100;
